LIN {X 0,Y 523.945,Z 504.224,A -85,B 0,C 180,E1 -4885.419,E2 -4885.419} C_VEL
LIN {X 0,Y 523.961,Z 504.216,A -85,B 0,C 180,E1 -4887.999,E2 -4887.999} C_VEL
LIN {X 0,Y 523.943,Z 504.222,A -85,B 0,C 180,E1 -4890.857,E2 -4890.857} C_VEL
LIN {X 0,Y 524,Z 504.295,A -85,B 0,C 180,E1 -4893.743,E2 -4893.743} C_VEL
LIN {X 0,Y 524.381,Z 507.648,A -85,B 0,C 180,E1 -4894.482,E2 -4894.482} C_VEL
LIN {X 0,Y 524.137,Z 518.874,A -85,B 0,C 180,E1 -4896.905,E2 -4896.905} C_VEL
LIN {X 0,Y 525.983,Z 529.654,A -85,B 0,C 180,E1 -4897.12,E2 -4897.12} C_VEL
LIN {X 0,Y 525.614,Z 604.892,A -85,B 0,C 180,E1 -4898.152,E2 -4898.152} C_VEL
LIN {X 0,Y 524.967,Z 610.73,A -85,B 0,C 180,E1 -4898.214,E2 -4898.214} C_VEL
LIN {X 0,Y 519.34,Z 629.652,A -85,B 0,C 180,E1 -4898.382,E2 -4898.382} C_VEL
LIN {X 0,Y 518.506,Z 635.385,A -85,B 0,C 180,E1 -4898.513,E2 -4898.513} C_VEL
LIN {X 0,Y 518.253,Z 648.027,A -85,B 0,C 180,E1 -4898.968,E2 -4898.968} C_VEL
LIN {X 0,Y 517.987,Z 659.606,A -85,B 0,C 180,E1 -4899.537,E2 -4899.537} C_VEL
LIN {X 0,Y 517.725,Z 670.589,A -85,B 0,C 180,E1 -4900.234,E2 -4900.234} C_VEL
LIN {X 0,Y 517.389,Z 681.214,A -85,B 0,C 180,E1 -4901.079,E2 -4901.079} C_VEL
LIN {X 0,Y 517.094,Z 690.566,A -85,B 0,C 180,E1 -4902.002,E2 -4902.002} C_VEL
LIN {X 0,Y 516.862,Z 699.506,A -85,B 0,C 180,E1 -4903.086,E2 -4903.086} C_VEL
LIN {X 0,Y 516.642,Z 706.907,A -85,B 0,C 180,E1 -4904.187,E2 -4904.187} C_VEL
LIN {X 0,Y 516.464,Z 714.132,A -85,B 0,C 180,E1 -4905.541,E2 -4905.541} C_VEL
LIN {X 0,Y 516.394,Z 718.741,A -85,B 0,C 180,E1 -4906.638,E2 -4906.638} C_VEL
LIN {X 0,Y 516.329,Z 722.395,A -85,B 0,C 180,E1 -4907.739,E2 -4907.739} C_VEL
LIN {X 0,Y 516.211,Z 725.817,A -85,B 0,C 180,E1 -4909.195,E2 -4909.195} C_VEL
LIN {X 0,Y 516.162,Z 727.383,A -85,B 0,C 180,E1 -4910.213,E2 -4910.213} C_VEL
LIN {X 0,Y 516.132,Z 728.224,A -85,B 0,C 180,E1 -4911.219,E2 -4911.219} C_VEL
LIN {X 0,Y 516.157,Z 728.432,A -85,B 0,C 180,E1 -4912.215,E2 -4912.215} C_VEL
LIN {X 0,Y 516.162,Z 727.807,A -85,B 0,C 180,E1 -4913.449,E2 -4913.449} C_VEL
LIN {X 0,Y 516.18,Z 726.02,A -85,B 0,C 180,E1 -4914.777,E2 -4914.777} C_VEL
LIN {X 0,Y 516.291,Z 722.961,A -85,B 0,C 180,E1 -4916.135,E2 -4916.135} C_VEL
LIN {X 0,Y 516.389,Z 718.385,A -85,B 0,C 180,E1 -4917.544,E2 -4917.544} C_VEL
LIN {X 0,Y 516.513,Z 712.566,A -85,B 0,C 180,E1 -4918.866,E2 -4918.866} C_VEL
LIN {X 0,Y 516.728,Z 705.121,A -85,B 0,C 180,E1 -4920.183,E2 -4920.183} C_VEL
LIN {X 0,Y 516.932,Z 696.702,A -85,B 0,C 180,E1 -4921.365,E2 -4921.365} C_VEL
LIN {X 0,Y 517.239,Z 686.68,A -85,B 0,C 180,E1 -4922.486,E2 -4922.486} C_VEL
LIN {X 0,Y 517.514,Z 676.852,A -85,B 0,C 180,E1 -4923.376,E2 -4923.376} C_VEL
LIN {X 0,Y 517.839,Z 665.892,A -85,B 0,C 180,E1 -4924.17,E2 -4924.17} C_VEL
LIN {X 0,Y 518.14,Z 653.517,A -85,B 0,C 180,E1 -4924.868,E2 -4924.868} C_VEL
LIN {X 0,Y 518.396,Z 641.103,A -85,B 0,C 180,E1 -4925.39,E2 -4925.39} C_VEL
LIN {X 0,Y 518.587,Z 628.298,A -85,B 0,C 180,E1 -4925.757,E2 -4925.757} C_VEL
LIN {X 0,Y 518.739,Z 608.806,A -85,B 0,C 180,E1 -4926.072,E2 -4926.072} C_VEL
LIN {X 0,Y 519.065,Z 529.137,A -85,B 0,C 180,E1 -4927.182,E2 -4927.182} C_VEL
LIN {X 0,Y 517.13,Z 519.018,A -85,B 0,C 180,E1 -4927.402,E2 -4927.402} C_VEL
LIN {X 0,Y 517.309,Z 507.574,A -85,B 0,C 180,E1 -4929.877,E2 -4929.877} C_VEL
LIN {X 0,Y 516.971,Z 505.092,A -85,B 0,C 180,E1 -4930.442,E2 -4930.442} C_VEL
LIN {X 0,Y 516.911,Z 505.095,A -85,B 0,C 180,E1 -4933.411,E2 -4933.411} C_VEL
LIN {X 0,Y 516.892,Z 505.093,A -85,B 0,C 180,E1 -4935.834,E2 -4935.834} C_VEL
LIN {X 0,Y 516.962,Z 505.086,A -85,B 0,C 180,E1 -4938.234,E2 -4938.234} C_VEL
LIN {X 0,Y 516.966,Z 505.086,A -85,B 0,C 180,E1 -4941.4,E2 -4941.4} C_VEL
LIN {X 0,Y 517,Z 505.08,A -85,B 0,C 180,E1 -4943.757,E2 -4943.757} C_VEL
LIN {X 0,Y 517.012,Z 505.088,A -85,B 0,C 180,E1 -4946.883,E2 -4946.883} C_VEL
LIN {X 0,Y 517.083,Z 505.069,A -85,B 0,C 180,E1 -4950,E2 -4950} C_VEL
LIN {X 0,Y 517.011,Z 505.085,A -85,B 0,C 180,E1 -4953.117,E2 -4953.117} C_VEL
LIN {X 0,Y 517.013,Z 505.079,A -85,B 0,C 180,E1 -4956.243,E2 -4956.243} C_VEL
LIN {X 0,Y 516.952,Z 505.089,A -85,B 0,C 180,E1 -4959.389,E2 -4959.389} C_VEL
LIN {X 0,Y 516.95,Z 505.086,A -85,B 0,C 180,E1 -4961.807,E2 -4961.807} C_VEL
LIN {X 0,Y 516.941,Z 505.094,A -85,B 0,C 180,E1 -4965.146,E2 -4965.146} C_VEL
LIN {X 0,Y 516.923,Z 505.09,A -85,B 0,C 180,E1 -4968.222,E2 -4968.222} C_VEL
LIN {X 0,Y 516.909,Z 505.096,A -85,B 0,C 180,E1 -4970.701,E2 -4970.701} C_VEL
LIN {X 0,Y 516.907,Z 505.091,A -85,B 0,C 180,E1 -4974.072,E2 -4974.072} C_VEL
LIN {X 0,Y 516.922,Z 505.094,A -85,B 0,C 180,E1 -4976.657,E2 -4976.657} C_VEL
LIN {X 0,Y 516.92,Z 505.092,A -85,B 0,C 180,E1 -4979.526,E2 -4979.526} C_VEL
LIN {X 0,Y 516.895,Z 505.095,A -85,B 0,C 180,E1 -4982.544,E2 -4982.544} C_VEL
LIN {X 0,Y 516.877,Z 505.1,A -85,B 0,C 180,E1 -4985.332,E2 -4985.332} C_VEL
LIN {X 0,Y 516.879,Z 505.095,A -85,B 0,C 180,E1 -4987.944,E2 -4987.944} C_VEL
LIN {X 0,Y 516.902,Z 505.097,A -85,B 0,C 180,E1 -4990.739,E2 -4990.739} C_VEL
LIN {X 0,Y 516.876,Z 505.095,A -85,B 0,C 180,E1 -4993.903,E2 -4993.903} C_VEL
LIN {X 0,Y 516.874,Z 505.095,A -85,B 0,C 180,E1 -4996.106,E2 -4996.106} C_VEL
LIN {X 0,Y 516.896,Z 505.099,A -85,B 0,C 180,E1 -4999.26,E2 -4999.26} C_VEL
LIN {X 0,Y 516.877,Z 505.095,A -85,B 0,C 180,E1 -5002.056,E2 -5002.056} C_VEL
LIN {X 0,Y 516.888,Z 505.102,A -85,B 0,C 180,E1 -5005.176,E2 -5005.176} C_VEL
LIN {X 0,Y 516.873,Z 505.096,A -85,B 0,C 180,E1 -5007.976,E2 -5007.976} C_VEL
LIN {X 0,Y 516.926,Z 505.092,A -85,B 0,C 180,E1 -5010.696,E2 -5010.696} C_VEL
LIN {X 0,Y 516.935,Z 505.089,A -85,B 0,C 180,E1 -5013.803,E2 -5013.803} C_VEL
LIN {X 0,Y 516.862,Z 505.101,A -85,B 0,C 180,E1 -5016.777,E2 -5016.777} C_VEL
LIN {X 0,Y 516.929,Z 505.09,A -85,B 0,C 180,E1 -5019.731,E2 -5019.731} C_VEL
LIN {X 0,Y 516.921,Z 505.091,A -85,B 0,C 180,E1 -5022.596,E2 -5022.596} C_VEL
LIN {X 0,Y 516.931,Z 505.096,A -85,B 0,C 180,E1 -5025.03,E2 -5025.03} C_VEL
LIN {X 0,Y 516.994,Z 505.081,A -85,B 0,C 180,E1 -5028.235,E2 -5028.235} C_VEL
LIN {X 0,Y 516.963,Z 505.09,A -85,B 0,C 180,E1 -5031.4,E2 -5031.4} C_VEL
LIN {X 0,Y 517.055,Z 505.074,A -85,B 0,C 180,E1 -5034.541,E2 -5034.541} C_VEL
LIN {X 0,Y 517.075,Z 505.073,A -85,B 0,C 180,E1 -5037.663,E2 -5037.663} C_VEL
LIN {X 0,Y 517.087,Z 505.072,A -85,B 0,C 180,E1 -5040.779,E2 -5040.779} C_VEL
LIN {X 0,Y 517.036,Z 505.083,A -85,B 0,C 180,E1 -5043.117,E2 -5043.117} C_VEL
LIN {X 0,Y 517.007,Z 505.079,A -85,B 0,C 180,E1 -5046.244,E2 -5046.244} C_VEL
LIN {X 0,Y 516.951,Z 505.093,A -85,B 0,C 180,E1 -5049.39,E2 -5049.39} C_VEL
LIN {X 0,Y 516.948,Z 505.088,A -85,B 0,C 180,E1 -5051.811,E2 -5051.811} C_VEL
LIN {X 0,Y 516.935,Z 505.096,A -85,B 0,C 180,E1 -5055.147,E2 -5055.147} C_VEL
LIN {X 0,Y 516.918,Z 505.09,A -85,B 0,C 180,E1 -5058.223,E2 -5058.223} C_VEL
LIN {X 0,Y 516.905,Z 505.093,A -85,B 0,C 180,E1 -5060.702,E2 -5060.702} C_VEL
LIN {X 0,Y 516.904,Z 505.092,A -85,B 0,C 180,E1 -5064.073,E2 -5064.073} C_VEL
LIN {X 0,Y 516.923,Z 505.091,A -85,B 0,C 180,E1 -5066.658,E2 -5066.658} C_VEL
LIN {X 0,Y 516.918,Z 505.096,A -85,B 0,C 180,E1 -5069.527,E2 -5069.527} C_VEL
LIN {X 0,Y 516.895,Z 505.093,A -85,B 0,C 180,E1 -5072.545,E2 -5072.545} C_VEL
LIN {X 0,Y 516.879,Z 505.104,A -85,B 0,C 180,E1 -5075.333,E2 -5075.333} C_VEL
LIN {X 0,Y 516.88,Z 505.096,A -85,B 0,C 180,E1 -5077.945,E2 -5077.945} C_VEL
LIN {X 0,Y 516.882,Z 505.096,A -85,B 0,C 180,E1 -5080.742,E2 -5080.742} C_VEL
LIN {X 0,Y 516.901,Z 505.094,A -85,B 0,C 180,E1 -5082.83,E2 -5082.83} C_VEL
LIN {X 0,Y 516.919,Z 505.094,A -85,B 0,C 180,E1 -5085.011,E2 -5085.011} C_VEL
LIN {X 0,Y 516.921,Z 505.09,A -85,B 0,C 180,E1 -5088.398,E2 -5088.398} C_VEL
LIN {X 0,Y 516.885,Z 505.102,A -85,B 0,C 180,E1 -5091.286,E2 -5091.286} C_VEL
LIN {X 0,Y 516.886,Z 505.094,A -85,B 0,C 180,E1 -5094.222,E2 -5094.222} C_VEL
LIN {X 0,Y 516.897,Z 505.098,A -85,B 0,C 180,E1 -5097.054,E2 -5097.054} C_VEL
LIN {X 0,Y 516.893,Z 505.099,A -85,B 0,C 180,E1 -5099.797,E2 -5099.797} C_VEL
LIN {X 0,Y 516.928,Z 505.092,A -85,B 0,C 180,E1 -5102.468,E2 -5102.468} C_VEL
LIN {X 0,Y 516.976,Z 505.23,A -85,B 0,C 180,E1 -5104.241,E2 -5104.241} C_VEL
LIN {X 0,Y 518.814,Z 514.974,A -85,B 0,C 180,E1 -5105.835,E2 -5105.835} C_VEL
LIN {X 0,Y 518.489,Z 528.641,A -85,B 0,C 180,E1 -5107.905,E2 -5107.905} C_VEL
LIN {X 0,Y 517.995,Z 548.15,A -85,B 0,C 180,E1 -5110.791,E2 -5110.791} C_VEL
LIN {X 0,Y 517.507,Z 568.945,A -85,B 0,C 180,E1 -5113.836,E2 -5113.836} C_VEL
LIN {X 0,Y 517.393,Z 574.378,A -85,B 0,C 180,E1 -5114.63,E2 -5114.63} C_VEL
LIN {X 0,Y 519.12,Z 586.795,A -85,B 0,C 180,E1 -5114.861,E2 -5114.861} C_VEL
LIN {X 0,Y 518.584,Z 682.754,A -85,B 0,C 180,E1 -5116.206,E2 -5116.206} C_VEL
LIN {X 0,Y 518.371,Z 696.184,A -85,B 0,C 180,E1 -5116.55,E2 -5116.55} C_VEL
LIN {X 0,Y 518.095,Z 709.57,A -85,B 0,C 180,E1 -5117.067,E2 -5117.067} C_VEL
LIN {X 0,Y 517.846,Z 721.086,A -85,B 0,C 180,E1 -5117.675,E2 -5117.675} C_VEL
LIN {X 0,Y 517.534,Z 732.47,A -85,B 0,C 180,E1 -5118.446,E2 -5118.446} C_VEL
LIN {X 0,Y 517.2,Z 742.972,A -85,B 0,C 180,E1 -5119.331,E2 -5119.331} C_VEL
LIN {X 0,Y 516.993,Z 751.565,A -85,B 0,C 180,E1 -5120.217,E2 -5120.217} C_VEL
LIN {X 0,Y 516.763,Z 759.494,A -85,B 0,C 180,E1 -5121.199,E2 -5121.199} C_VEL
LIN {X 0,Y 516.563,Z 767.24,A -85,B 0,C 180,E1 -5122.377,E2 -5122.377} C_VEL
LIN {X 0,Y 516.427,Z 774.381,A -85,B 0,C 180,E1 -5123.75,E2 -5123.75} C_VEL
LIN {X 0,Y 516.314,Z 779.131,A -85,B 0,C 180,E1 -5124.924,E2 -5124.924} C_VEL
LIN {X 0,Y 516.355,Z 782.768,A -85,B 0,C 180,E1 -5126.098,E2 -5126.098} C_VEL
LIN {X 0,Y 516.283,Z 784.638,A -85,B 0,C 180,E1 -5126.879,E2 -5126.879} C_VEL
LIN {X 0,Y 516.26,Z 786.042,A -85,B 0,C 180,E1 -5127.659,E2 -5127.659} C_VEL
LIN {X 0,Y 516.16,Z 787.651,A -85,B 0,C 180,E1 -5129.22,E2 -5129.22} C_VEL
LIN {X 0,Y 516.154,Z 787.868,A -85,B 0,C 180,E1 -5130,E2 -5130} C_VEL
LIN {X 0,Y 516.192,Z 787.042,A -85,B 0,C 180,E1 -5131.56,E2 -5131.56} C_VEL
LIN {X 0,Y 516.26,Z 786.043,A -85,B 0,C 180,E1 -5132.341,E2 -5132.341} C_VEL
LIN {X 0,Y 516.283,Z 784.638,A -85,B 0,C 180,E1 -5133.121,E2 -5133.121} C_VEL
LIN {X 0,Y 516.326,Z 781.683,A -85,B 0,C 180,E1 -5134.293,E2 -5134.293} C_VEL
LIN {X 0,Y 516.384,Z 777.682,A -85,B 0,C 180,E1 -5135.467,E2 -5135.467} C_VEL
LIN {X 0,Y 516.444,Z 772.354,A -85,B 0,C 180,E1 -5136.678,E2 -5136.678} C_VEL
LIN {X 0,Y 516.579,Z 766.048,A -85,B 0,C 180,E1 -5137.819,E2 -5137.819} C_VEL
LIN {X 0,Y 516.809,Z 757.966,A -85,B 0,C 180,E1 -5138.997,E2 -5138.997} C_VEL
LIN {X 0,Y 517.021,Z 749.729,A -85,B 0,C 180,E1 -5139.98,E2 -5139.98} C_VEL
LIN {X 0,Y 517.313,Z 739.687,A -85,B 0,C 180,E1 -5140.964,E2 -5140.964} C_VEL
LIN {X 0,Y 517.631,Z 728.435,A -85,B 0,C 180,E1 -5141.844,E2 -5141.844} C_VEL
LIN {X 0,Y 517.942,Z 717.243,A -85,B 0,C 180,E1 -5142.539,E2 -5142.539} C_VEL
LIN {X 0,Y 518.198,Z 704.93,A -85,B 0,C 180,E1 -5143.13,E2 -5143.13} C_VEL
LIN {X 0,Y 518.447,Z 691.96,A -85,B 0,C 180,E1 -5143.573,E2 -5143.573} C_VEL
LIN {X 0,Y 518.654,Z 679.665,A -85,B 0,C 180,E1 -5143.842,E2 -5143.842} C_VEL
LIN {X 0,Y 519.042,Z 585.382,A -85,B 0,C 180,E1 -5145.159,E2 -5145.159} C_VEL
LIN {X 0,Y 517.381,Z 574.125,A -85,B 0,C 180,E1 -5145.38,E2 -5145.38} C_VEL
LIN {X 0,Y 517.857,Z 552.08,A -85,B 0,C 180,E1 -5148.597,E2 -5148.597} C_VEL
LIN {X 0,Y 518.397,Z 531.131,A -85,B 0,C 180,E1 -5151.68,E2 -5151.68} C_VEL
LIN {X 0,Y 518.776,Z 515.802,A -85,B 0,C 180,E1 -5153.979,E2 -5153.979} C_VEL
LIN {X 0,Y 518.207,Z 511.389,A -85,B 0,C 180,E1 -5154.678,E2 -5154.678} C_VEL
LIN {X 0,Y 516.955,Z 505.092,A -85,B 0,C 180,E1 -5155.733,E2 -5155.733} C_VEL
LIN {X 0,Y 516.92,Z 505.098,A -85,B 0,C 180,E1 -5158.414,E2 -5158.414} C_VEL
LIN {X 0,Y 516.891,Z 505.099,A -85,B 0,C 180,E1 -5161.109,E2 -5161.109} C_VEL
LIN {X 0,Y 516.912,Z 505.095,A -85,B 0,C 180,E1 -5163.966,E2 -5163.966} C_VEL
LIN {X 0,Y 516.882,Z 505.104,A -85,B 0,C 180,E1 -5166.745,E2 -5166.745} C_VEL
LIN {X 0,Y 516.901,Z 505.093,A -85,B 0,C 180,E1 -5169.718,E2 -5169.718} C_VEL
LIN {X 0,Y 516.904,Z 505.1,A -85,B 0,C 180,E1 -5172.76,E2 -5172.76} C_VEL
LIN {X 0,Y 516.919,Z 505.095,A -85,B 0,C 180,E1 -5175.009,E2 -5175.009} C_VEL
LIN {X 0,Y 516.913,Z 505.094,A -85,B 0,C 180,E1 -5178.397,E2 -5178.397} C_VEL
LIN {X 0,Y 516.879,Z 505.098,A -85,B 0,C 180,E1 -5181.284,E2 -5181.284} C_VEL
LIN {X 0,Y 516.886,Z 505.096,A -85,B 0,C 180,E1 -5184.22,E2 -5184.22} C_VEL
LIN {X 0,Y 516.893,Z 505.099,A -85,B 0,C 180,E1 -5187.052,E2 -5187.052} C_VEL
LIN {X 0,Y 516.896,Z 505.093,A -85,B 0,C 180,E1 -5189.796,E2 -5189.796} C_VEL
LIN {X 0,Y 516.924,Z 505.093,A -85,B 0,C 180,E1 -5192.467,E2 -5192.467} C_VEL
LIN {X 0,Y 516.905,Z 505.096,A -85,B 0,C 180,E1 -5195.071,E2 -5195.071} C_VEL
LIN {X 0,Y 516.879,Z 505.099,A -85,B 0,C 180,E1 -5198.462,E2 -5198.462} C_VEL
LIN {X 0,Y 516.9,Z 505.101,A -85,B 0,C 180,E1 -5200.954,E2 -5200.954} C_VEL
LIN {X 0,Y 516.909,Z 505.094,A -85,B 0,C 180,E1 -5203.41,E2 -5203.41} C_VEL
LIN {X 0,Y 516.886,Z 505.094,A -85,B 0,C 180,E1 -5205.833,E2 -5205.833} C_VEL
LIN {X 0,Y 516.956,Z 505.087,A -85,B 0,C 180,E1 -5208.233,E2 -5208.233} C_VEL
LIN {X 0,Y 516.964,Z 505.088,A -85,B 0,C 180,E1 -5211.399,E2 -5211.399} C_VEL
LIN {X 0,Y 517.055,Z 505.075,A -85,B 0,C 180,E1 -5214.54,E2 -5214.54} C_VEL
LIN {X 0,Y 517.075,Z 505.072,A -85,B 0,C 180,E1 -5217.663,E2 -5217.663} C_VEL
LIN {X 0,Y 517.087,Z 505.074,A -85,B 0,C 180,E1 -5220.778,E2 -5220.778} C_VEL
LIN {X 0,Y 517.01,Z 505.086,A -85,B 0,C 180,E1 -5223.117,E2 -5223.117} C_VEL
LIN {X 0,Y 517.006,Z 505.079,A -85,B 0,C 180,E1 -5226.243,E2 -5226.243} C_VEL
LIN {X 0,Y 516.949,Z 505.092,A -85,B 0,C 180,E1 -5229.389,E2 -5229.389} C_VEL
LIN {X 0,Y 516.947,Z 505.088,A -85,B 0,C 180,E1 -5231.81,E2 -5231.81} C_VEL
LIN {X 0,Y 516.933,Z 505.097,A -85,B 0,C 180,E1 -5235.146,E2 -5235.146} C_VEL
LIN {X 0,Y 516.917,Z 505.091,A -85,B 0,C 180,E1 -5238.222,E2 -5238.222} C_VEL
LIN {X 0,Y 516.903,Z 505.096,A -85,B 0,C 180,E1 -5240.701,E2 -5240.701} C_VEL
LIN {X 0,Y 516.901,Z 505.095,A -85,B 0,C 180,E1 -5244.072,E2 -5244.072} C_VEL
LIN {X 0,Y 516.92,Z 505.096,A -85,B 0,C 180,E1 -5246.658,E2 -5246.658} C_VEL
LIN {X 0,Y 516.915,Z 505.098,A -85,B 0,C 180,E1 -5249.527,E2 -5249.527} C_VEL
LIN {X 0,Y 516.894,Z 505.099,A -85,B 0,C 180,E1 -5252.545,E2 -5252.545} C_VEL
LIN {X 0,Y 516.929,Z 505.102,A -85,B 0,C 180,E1 -5253.584,E2 -5253.584} C_VEL
LIN {X 0,Y 517.389,Z 509.488,A -85,B 0,C 180,E1 -5254.565,E2 -5254.565} C_VEL
LIN {X 0,Y 517.176,Z 519.353,A -85,B 0,C 180,E1 -5256.703,E2 -5256.703} C_VEL
LIN {X 0,Y 519.152,Z 530.648,A -85,B 0,C 180,E1 -5256.928,E2 -5256.928} C_VEL
LIN {X 0,Y 518.613,Z 625.517,A -85,B 0,C 180,E1 -5258.271,E2 -5258.271} C_VEL
LIN {X 0,Y 518.506,Z 635.385,A -85,B 0,C 180,E1 -5258.513,E2 -5258.513} C_VEL
LIN {X 0,Y 517.638,Z 641.076,A -85,B 0,C 180,E1 -5258.669,E2 -5258.669} C_VEL
LIN {X 0,Y 514.689,Z 650.202,A -85,B 0,C 180,E1 -5258.953,E2 -5258.953} C_VEL
LIN {X 0,Y 511.77,Z 659.029,A -85,B 0,C 180,E1 -5259.327,E2 -5259.327} C_VEL
LIN {X 0,Y 510.95,Z 664.243,A -85,B 0,C 180,E1 -5259.62,E2 -5259.62} C_VEL
LIN {X 0,Y 510.627,Z 675.597,A -85,B 0,C 180,E1 -5260.423,E2 -5260.423} C_VEL
LIN {X 0,Y 510.328,Z 684.665,A -85,B 0,C 180,E1 -5261.216,E2 -5261.216} C_VEL
LIN {X 0,Y 510.034,Z 693.646,A -85,B 0,C 180,E1 -5262.167,E2 -5262.167} C_VEL
LIN {X 0,Y 509.742,Z 702.705,A -85,B 0,C 180,E1 -5263.358,E2 -5263.358} C_VEL
LIN {X 0,Y 509.546,Z 709.578,A -85,B 0,C 180,E1 -5264.475,E2 -5264.475} C_VEL
LIN {X 0,Y 509.393,Z 716.296,A -85,B 0,C 180,E1 -5265.842,E2 -5265.842} C_VEL
LIN {X 0,Y 509.305,Z 720.697,A -85,B 0,C 180,E1 -5267,E2 -5267} C_VEL
LIN {X 0,Y 509.203,Z 724.905,A -85,B 0,C 180,E1 -5268.511,E2 -5268.511} C_VEL
LIN {X 0,Y 509.11,Z 726.92,A -85,B 0,C 180,E1 -5269.549,E2 -5269.549} C_VEL
LIN {X 0,Y 509.071,Z 728.236,A -85,B 0,C 180,E1 -5270.633,E2 -5270.633} C_VEL
LIN {X 0,Y 509.068,Z 728.847,A -85,B 0,C 180,E1 -5271.898,E2 -5271.898} C_VEL
LIN {X 0,Y 509.072,Z 728.435,A -85,B 0,C 180,E1 -5273.198,E2 -5273.198} C_VEL
LIN {X 0,Y 509.086,Z 726.867,A -85,B 0,C 180,E1 -5274.563,E2 -5274.563} C_VEL
LIN {X 0,Y 509.191,Z 724.115,A -85,B 0,C 180,E1 -5275.907,E2 -5275.907} C_VEL
LIN {X 0,Y 509.285,Z 719.822,A -85,B 0,C 180,E1 -5277.328,E2 -5277.328} C_VEL
LIN {X 0,Y 509.465,Z 713.798,A -85,B 0,C 180,E1 -5278.79,E2 -5278.79} C_VEL
LIN {X 0,Y 509.637,Z 707.267,A -85,B 0,C 180,E1 -5280.008,E2 -5280.008} C_VEL
LIN {X 0,Y 509.848,Z 699.633,A -85,B 0,C 180,E1 -5281.155,E2 -5281.155} C_VEL
LIN {X 0,Y 510.148,Z 690.272,A -85,B 0,C 180,E1 -5282.294,E2 -5282.294} C_VEL
LIN {X 0,Y 510.475,Z 680.23,A -85,B 0,C 180,E1 -5283.273,E2 -5283.273} C_VEL
LIN {X 0,Y 510.806,Z 669.716,A -85,B 0,C 180,E1 -5284.098,E2 -5284.098} C_VEL
LIN {X 0,Y 511.11,Z 658.059,A -85,B 0,C 180,E1 -5284.826,E2 -5284.826} C_VEL
LIN {X 0,Y 511.386,Z 646.447,A -85,B 0,C 180,E1 -5285.38,E2 -5285.38} C_VEL
LIN {X 0,Y 511.613,Z 633.316,A -85,B 0,C 180,E1 -5285.825,E2 -5285.825} C_VEL
LIN {X 0,Y 511.807,Z 620.1,A -85,B 0,C 180,E1 -5286.104,E2 -5286.104} C_VEL
LIN {X 0,Y 512.161,Z 529.548,A -85,B 0,C 180,E1 -5287.39,E2 -5287.39} C_VEL
LIN {X 0,Y 510.139,Z 519.449,A -85,B 0,C 180,E1 -5287.609,E2 -5287.609} C_VEL
LIN {X 0,Y 510.336,Z 509.091,A -85,B 0,C 180,E1 -5289.862,E2 -5289.862} C_VEL
LIN {X 0,Y 509.896,Z 505.974,A -85,B 0,C 180,E1 -5290.579,E2 -5290.579} C_VEL
LIN {X 0,Y 509.881,Z 505.973,A -85,B 0,C 180,E1 -5293.175,E2 -5293.175} C_VEL
LIN {X 0,Y 509.861,Z 505.97,A -85,B 0,C 180,E1 -5295.634,E2 -5295.634} C_VEL
LIN {X 0,Y 509.899,Z 505.965,A -85,B 0,C 180,E1 -5298.123,E2 -5298.123} C_VEL
LIN {X 0,Y 509.912,Z 505.966,A -85,B 0,C 180,E1 -5301.28,E2 -5301.28} C_VEL
LIN {X 0,Y 509.951,Z 505.958,A -85,B 0,C 180,E1 -5303.67,E2 -5303.67} C_VEL
LIN {X 0,Y 509.954,Z 505.966,A -85,B 0,C 180,E1 -5306.84,E2 -5306.84} C_VEL
LIN {X 0,Y 510.061,Z 505.949,A -85,B 0,C 180,E1 -5309.211,E2 -5309.211} C_VEL
LIN {X 0,Y 510.054,Z 505.947,A -85,B 0,C 180,E1 -5312.369,E2 -5312.369} C_VEL
LIN {X 0,Y 509.98,Z 505.956,A -85,B 0,C 180,E1 -5316.329,E2 -5316.329} C_VEL
LIN {X 0,Y 509.914,Z 505.968,A -85,B 0,C 180,E1 -5318.72,E2 -5318.72} C_VEL
LIN {X 0,Y 509.901,Z 505.964,A -85,B 0,C 180,E1 -5321.931,E2 -5321.931} C_VEL
LIN {X 0,Y 509.89,Z 505.97,A -85,B 0,C 180,E1 -5325.242,E2 -5325.242} C_VEL
LIN {X 0,Y 509.885,Z 505.966,A -85,B 0,C 180,E1 -5328.001,E2 -5328.001} C_VEL
LIN {X 0,Y 509.846,Z 505.98,A -85,B 0,C 180,E1 -5331.001,E2 -5331.001} C_VEL
LIN {X 0,Y 509.832,Z 505.974,A -85,B 0,C 180,E1 -5333.563,E2 -5333.563} C_VEL
LIN {X 0,Y 509.907,Z 505.965,A -85,B 0,C 180,E1 -5336.378,E2 -5336.378} C_VEL
LIN {X 0,Y 509.881,Z 505.973,A -85,B 0,C 180,E1 -5338.843,E2 -5338.843} C_VEL
LIN {X 0,Y 509.821,Z 505.976,A -85,B 0,C 180,E1 -5341.589,E2 -5341.589} C_VEL
LIN {X 0,Y 509.847,Z 505.972,A -85,B 0,C 180,E1 -5344.413,E2 -5344.413} C_VEL
LIN {X 0,Y 509.816,Z 505.979,A -85,B 0,C 180,E1 -5347.34,E2 -5347.34} C_VEL
LIN {X 0,Y 509.856,Z 505.971,A -85,B 0,C 180,E1 -5350.379,E2 -5350.379} C_VEL
LIN {X 0,Y 509.834,Z 505.982,A -85,B 0,C 180,E1 -5353.064,E2 -5353.064} C_VEL
LIN {X 0,Y 509.822,Z 505.975,A -85,B 0,C 180,E1 -5355.792,E2 -5355.792} C_VEL
LIN {X 0,Y 509.857,Z 505.972,A -85,B 0,C 180,E1 -5358.575,E2 -5358.575} C_VEL
LIN {X 0,Y 509.849,Z 505.971,A -85,B 0,C 180,E1 -5361.785,E2 -5361.785} C_VEL
LIN {X 0,Y 509.838,Z 505.975,A -85,B 0,C 180,E1 -5364.623,E2 -5364.623} C_VEL
LIN {X 0,Y 509.857,Z 505.973,A -85,B 0,C 180,E1 -5367.481,E2 -5367.481} C_VEL
LIN {X 0,Y 509.872,Z 505.968,A -85,B 0,C 180,E1 -5370.269,E2 -5370.269} C_VEL
LIN {X 0,Y 509.878,Z 505.974,A -85,B 0,C 180,E1 -5372.944,E2 -5372.944} C_VEL
LIN {X 0,Y 509.861,Z 505.972,A -85,B 0,C 180,E1 -5375.574,E2 -5375.574} C_VEL
LIN {X 0,Y 509.812,Z 505.975,A -85,B 0,C 180,E1 -5378.149,E2 -5378.149} C_VEL
LIN {X 0,Y 509.855,Z 505.973,A -85,B 0,C 180,E1 -5380.682,E2 -5380.682} C_VEL
LIN {X 0,Y 509.877,Z 505.976,A -85,B 0,C 180,E1 -5383.175,E2 -5383.175} C_VEL
LIN {X 0,Y 509.854,Z 505.973,A -85,B 0,C 180,E1 -5385.634,E2 -5385.634} C_VEL
LIN {X 0,Y 509.919,Z 505.967,A -85,B 0,C 180,E1 -5388.875,E2 -5388.875} C_VEL
LIN {X 0,Y 509.942,Z 505.959,A -85,B 0,C 180,E1 -5392.079,E2 -5392.079} C_VEL
LIN {X 0,Y 510.001,Z 505.952,A -85,B 0,C 180,E1 -5394.465,E2 -5394.465} C_VEL
LIN {X 0,Y 510.046,Z 505.949,A -85,B 0,C 180,E1 -5397.631,E2 -5397.631} C_VEL
LIN {X 0,Y 510.057,Z 505.948,A -85,B 0,C 180,E1 -5400.79,E2 -5400.79} C_VEL
LIN {X 0,Y 509.977,Z 505.963,A -85,B 0,C 180,E1 -5403.16,E2 -5403.16} C_VEL
LIN {X 0,Y 509.974,Z 505.955,A -85,B 0,C 180,E1 -5406.33,E2 -5406.33} C_VEL
LIN {X 0,Y 509.911,Z 505.965,A -85,B 0,C 180,E1 -5408.721,E2 -5408.721} C_VEL
LIN {X 0,Y 509.896,Z 505.966,A -85,B 0,C 180,E1 -5411.932,E2 -5411.932} C_VEL
LIN {X 0,Y 509.885,Z 505.976,A -85,B 0,C 180,E1 -5415.242,E2 -5415.242} C_VEL
LIN {X 0,Y 509.88,Z 505.967,A -85,B 0,C 180,E1 -5418.002,E2 -5418.002} C_VEL
LIN {X 0,Y 509.843,Z 505.976,A -85,B 0,C 180,E1 -5421.002,E2 -5421.002} C_VEL
LIN {X 0,Y 509.829,Z 505.978,A -85,B 0,C 180,E1 -5423.564,E2 -5423.564} C_VEL
LIN {X 0,Y 509.907,Z 505.963,A -85,B 0,C 180,E1 -5426.38,E2 -5426.38} C_VEL
LIN {X 0,Y 509.879,Z 505.97,A -85,B 0,C 180,E1 -5428.844,E2 -5428.844} C_VEL
LIN {X 0,Y 509.821,Z 505.979,A -85,B 0,C 180,E1 -5431.591,E2 -5431.591} C_VEL
LIN {X 0,Y 509.849,Z 505.971,A -85,B 0,C 180,E1 -5434.414,E2 -5434.414} C_VEL
LIN {X 0,Y 509.817,Z 505.984,A -85,B 0,C 180,E1 -5437.341,E2 -5437.341} C_VEL
LIN {X 0,Y 509.834,Z 505.972,A -85,B 0,C 180,E1 -5440.383,E2 -5440.383} C_VEL
LIN {X 0,Y 509.836,Z 505.977,A -85,B 0,C 180,E1 -5443.065,E2 -5443.065} C_VEL
LIN {X 0,Y 509.828,Z 505.976,A -85,B 0,C 180,E1 -5445.793,E2 -5445.793} C_VEL
LIN {X 0,Y 509.863,Z 505.969,A -85,B 0,C 180,E1 -5448.576,E2 -5448.576} C_VEL
LIN {X 0,Y 509.851,Z 505.974,A -85,B 0,C 180,E1 -5451.787,E2 -5451.787} C_VEL
LIN {X 0,Y 509.842,Z 505.972,A -85,B 0,C 180,E1 -5454.624,E2 -5454.624} C_VEL
LIN {X 0,Y 509.866,Z 505.978,A -85,B 0,C 180,E1 -5457.482,E2 -5457.482} C_VEL
LIN {X 0,Y 509.859,Z 505.972,A -85,B 0,C 180,E1 -5460.274,E2 -5460.274} C_VEL
LIN {X 0,Y 509.886,Z 505.973,A -85,B 0,C 180,E1 -5462.945,E2 -5462.945} C_VEL
LIN {X 0,Y 509.937,Z 506.123,A -85,B 0,C 180,E1 -5464.051,E2 -5464.051} C_VEL
LIN {X 0,Y 511.851,Z 515.902,A -85,B 0,C 180,E1 -5465.675,E2 -5465.675} C_VEL
LIN {X 0,Y 511.614,Z 528.317,A -85,B 0,C 180,E1 -5467.593,E2 -5467.593} C_VEL
LIN {X 0,Y 511.018,Z 549.202,A -85,B 0,C 180,E1 -5470.727,E2 -5470.727} C_VEL
LIN {X 0,Y 510.454,Z 569.93,A -85,B 0,C 180,E1 -5473.812,E2 -5473.812} C_VEL
LIN {X 0,Y 510.365,Z 574.163,A -85,B 0,C 180,E1 -5474.419,E2 -5474.419} C_VEL
LIN {X 0,Y 512.249,Z 587.055,A -85,B 0,C 180,E1 -5474.663,E2 -5474.663} C_VEL
LIN {X 0,Y 511.688,Z 682.184,A -85,B 0,C 180,E1 -5476.016,E2 -5476.016} C_VEL
LIN {X 0,Y 511.45,Z 695.682,A -85,B 0,C 180,E1 -5476.365,E2 -5476.365} C_VEL
LIN {X 0,Y 511.164,Z 709.095,A -85,B 0,C 180,E1 -5476.888,E2 -5476.888} C_VEL
LIN {X 0,Y 510.866,Z 720.898,A -85,B 0,C 180,E1 -5477.521,E2 -5477.521} C_VEL
LIN {X 0,Y 510.53,Z 732.026,A -85,B 0,C 180,E1 -5478.285,E2 -5478.285} C_VEL
LIN {X 0,Y 510.217,Z 742.539,A -85,B 0,C 180,E1 -5479.183,E2 -5479.183} C_VEL
LIN {X 0,Y 509.929,Z 751.135,A -85,B 0,C 180,E1 -5480.08,E2 -5480.08} C_VEL
LIN {X 0,Y 509.708,Z 759.071,A -85,B 0,C 180,E1 -5481.077,E2 -5481.077} C_VEL
LIN {X 0,Y 509.486,Z 766.823,A -85,B 0,C 180,E1 -5482.271,E2 -5482.271} C_VEL
LIN {X 0,Y 509.325,Z 773.967,A -85,B 0,C 180,E1 -5483.662,E2 -5483.662} C_VEL
LIN {X 0,Y 509.245,Z 778.723,A -85,B 0,C 180,E1 -5484.853,E2 -5484.853} C_VEL
LIN {X 0,Y 509.266,Z 782.36,A -85,B 0,C 180,E1 -5486.043,E2 -5486.043} C_VEL
LIN {X 0,Y 509.201,Z 784.232,A -85,B 0,C 180,E1 -5486.835,E2 -5486.835} C_VEL
LIN {X 0,Y 509.189,Z 785.637,A -85,B 0,C 180,E1 -5487.627,E2 -5487.627} C_VEL
LIN {X 0,Y 509.073,Z 787.245,A -85,B 0,C 180,E1 -5489.209,E2 -5489.209} C_VEL
LIN {X 0,Y 509.066,Z 787.461,A -85,B 0,C 180,E1 -5490,E2 -5490} C_VEL
LIN {X 0,Y 509.112,Z 786.632,A -85,B 0,C 180,E1 -5491.582,E2 -5491.582} C_VEL
LIN {X 0,Y 509.189,Z 785.632,A -85,B 0,C 180,E1 -5492.373,E2 -5492.373} C_VEL
LIN {X 0,Y 509.201,Z 784.222,A -85,B 0,C 180,E1 -5493.165,E2 -5493.165} C_VEL
LIN {X 0,Y 509.218,Z 781.261,A -85,B 0,C 180,E1 -5494.353,E2 -5494.353} C_VEL
LIN {X 0,Y 509.305,Z 777.256,A -85,B 0,C 180,E1 -5495.543,E2 -5495.543} C_VEL
LIN {X 0,Y 509.396,Z 771.55,A -85,B 0,C 180,E1 -5496.844,E2 -5496.844} C_VEL
LIN {X 0,Y 509.538,Z 764.361,A -85,B 0,C 180,E1 -5498.127,E2 -5498.127} C_VEL
LIN {X 0,Y 509.775,Z 756.01,A -85,B 0,C 180,E1 -5499.322,E2 -5499.322} C_VEL
LIN {X 0,Y 510.018,Z 747.449,A -85,B 0,C 180,E1 -5500.319,E2 -5500.319} C_VEL
LIN {X 0,Y 510.427,Z 736.883,A -85,B 0,C 180,E1 -5501.315,E2 -5501.315} C_VEL
LIN {X 0,Y 510.691,Z 726.091,A -85,B 0,C 180,E1 -5502.137,E2 -5502.137} C_VEL
LIN {X 0,Y 511.015,Z 714.956,A -85,B 0,C 180,E1 -5502.813,E2 -5502.813} C_VEL
LIN {X 0,Y 511.329,Z 703.15,A -85,B 0,C 180,E1 -5503.36,E2 -5503.36} C_VEL
LIN {X 0,Y 511.545,Z 689.542,A -85,B 0,C 180,E1 -5503.81,E2 -5503.81} C_VEL
LIN {X 0,Y 511.78,Z 675.86,A -85,B 0,C 180,E1 -5504.082,E2 -5504.082} C_VEL
LIN {X 0,Y 512.112,Z 585.715,A -85,B 0,C 180,E1 -5505.357,E2 -5505.357} C_VEL
LIN {X 0,Y 510.361,Z 573.691,A -85,B 0,C 180,E1 -5505.594,E2 -5505.594} C_VEL
LIN {X 0,Y 510.888,Z 551.622,A -85,B 0,C 180,E1 -5508.861,E2 -5508.861} C_VEL
LIN {X 0,Y 511.437,Z 532.12,A -85,B 0,C 180,E1 -5511.778,E2 -5511.778} C_VEL
LIN {X 0,Y 511.846,Z 516.823,A -85,B 0,C 180,E1 -5514.109,E2 -5514.109} C_VEL
LIN {X 0,Y 510.396,Z 508.38,A -85,B 0,C 180,E1 -5515.486,E2 -5515.486} C_VEL
LIN {X 0,Y 509.926,Z 505.968,A -85,B 0,C 180,E1 -5515.895,E2 -5515.895} C_VEL
LIN {X 0,Y 509.877,Z 505.974,A -85,B 0,C 180,E1 -5518.843,E2 -5518.843} C_VEL
LIN {X 0,Y 509.825,Z 505.977,A -85,B 0,C 180,E1 -5521.589,E2 -5521.589} C_VEL
LIN {X 0,Y 509.853,Z 505.98,A -85,B 0,C 180,E1 -5524.412,E2 -5524.412} C_VEL
LIN {X 0,Y 509.818,Z 505.977,A -85,B 0,C 180,E1 -5527.34,E2 -5527.34} C_VEL
LIN {X 0,Y 509.859,Z 505.975,A -85,B 0,C 180,E1 -5530.379,E2 -5530.379} C_VEL
LIN {X 0,Y 509.837,Z 505.977,A -85,B 0,C 180,E1 -5533.063,E2 -5533.063} C_VEL
LIN {X 0,Y 509.827,Z 505.974,A -85,B 0,C 180,E1 -5535.791,E2 -5535.791} C_VEL
LIN {X 0,Y 509.855,Z 505.976,A -85,B 0,C 180,E1 -5538.574,E2 -5538.574} C_VEL
LIN {X 0,Y 509.848,Z 505.971,A -85,B 0,C 180,E1 -5541.785,E2 -5541.785} C_VEL
LIN {X 0,Y 509.842,Z 505.978,A -85,B 0,C 180,E1 -5544.622,E2 -5544.622} C_VEL
LIN {X 0,Y 509.86,Z 505.971,A -85,B 0,C 180,E1 -5547.48,E2 -5547.48} C_VEL
LIN {X 0,Y 509.875,Z 505.969,A -85,B 0,C 180,E1 -5550.268,E2 -5550.268} C_VEL
LIN {X 0,Y 509.881,Z 505.975,A -85,B 0,C 180,E1 -5552.944,E2 -5552.944} C_VEL
LIN {X 0,Y 509.863,Z 505.968,A -85,B 0,C 180,E1 -5555.573,E2 -5555.573} C_VEL
LIN {X 0,Y 509.843,Z 505.977,A -85,B 0,C 180,E1 -5558.998,E2 -5558.998} C_VEL
LIN {X 0,Y 509.88,Z 505.967,A -85,B 0,C 180,E1 -5561.998,E2 -5561.998} C_VEL
LIN {X 0,Y 509.901,Z 505.972,A -85,B 0,C 180,E1 -5564.818,E2 -5564.818} C_VEL
LIN {X 0,Y 509.897,Z 505.965,A -85,B 0,C 180,E1 -5568.12,E2 -5568.12} C_VEL
LIN {X 0,Y 509.91,Z 505.968,A -85,B 0,C 180,E1 -5571.279,E2 -5571.279} C_VEL
LIN {X 0,Y 509.973,Z 505.955,A -85,B 0,C 180,E1 -5573.67,E2 -5573.67} C_VEL
LIN {X 0,Y 509.951,Z 505.965,A -85,B 0,C 180,E1 -5576.839,E2 -5576.839} C_VEL
LIN {X 0,Y 510.057,Z 505.95,A -85,B 0,C 180,E1 -5579.21,E2 -5579.21} C_VEL
LIN {X 0,Y 510.046,Z 505.948,A -85,B 0,C 180,E1 -5582.369,E2 -5582.369} C_VEL
LIN {X 0,Y 510.002,Z 505.954,A -85,B 0,C 180,E1 -5585.535,E2 -5585.535} C_VEL
LIN {X 0,Y 509.942,Z 505.96,A -85,B 0,C 180,E1 -5587.921,E2 -5587.921} C_VEL
LIN {X 0,Y 509.908,Z 505.971,A -85,B 0,C 180,E1 -5591.125,E2 -5591.125} C_VEL
LIN {X 0,Y 509.854,Z 505.972,A -85,B 0,C 180,E1 -5594.366,E2 -5594.366} C_VEL
LIN {X 0,Y 509.893,Z 505.969,A -85,B 0,C 180,E1 -5597.651,E2 -5597.651} C_VEL
LIN {X 0,Y 509.876,Z 505.969,A -85,B 0,C 180,E1 -5600.402,E2 -5600.402} C_VEL
LIN {X 0,Y 509.826,Z 505.98,A -85,B 0,C 180,E1 -5603.563,E2 -5603.563} C_VEL
LIN {X 0,Y 509.904,Z 505.969,A -85,B 0,C 180,E1 -5606.379,E2 -5606.379} C_VEL
LIN {X 0,Y 509.876,Z 505.975,A -85,B 0,C 180,E1 -5608.844,E2 -5608.844} C_VEL
LIN {X 0,Y 509.818,Z 505.983,A -85,B 0,C 180,E1 -5611.59,E2 -5611.59} C_VEL
LIN {X 0,Y 509.896,Z 506.076,A -85,B 0,C 180,E1 -5613.458,E2 -5613.458} C_VEL
LIN {X 0,Y 510.416,Z 511.163,A -85,B 0,C 180,E1 -5614.609,E2 -5614.609} C_VEL
LIN {X 0,Y 510.219,Z 519.801,A -85,B 0,C 180,E1 -5616.489,E2 -5616.489} C_VEL
LIN {X 0,Y 512.301,Z 530.6,A -85,B 0,C 180,E1 -5616.716,E2 -5616.716} C_VEL
LIN {X 0,Y 511.74,Z 625.853,A -85,B 0,C 180,E1 -5618.084,E2 -5618.084} C_VEL
LIN {X 0,Y 511.498,Z 639.488,A -85,B 0,C 180,E1 -5618.449,E2 -5618.449} C_VEL
LIN {X 0,Y 511.303,Z 652.192,A -85,B 0,C 180,E1 -5618.96,E2 -5618.96} C_VEL
LIN {X 0,Y 510.95,Z 664.243,A -85,B 0,C 180,E1 -5619.62,E2 -5619.62} C_VEL
LIN {X 0,Y 510.098,Z 669.438,A -85,B 0,C 180,E1 -5619.942,E2 -5619.942} C_VEL
LIN {X 0,Y 507.034,Z 677.595,A -85,B 0,C 180,E1 -5620.486,E2 -5620.486} C_VEL
LIN {X 0,Y 504.004,Z 685.249,A -85,B 0,C 180,E1 -5621.101,E2 -5621.101} C_VEL
LIN {X 0,Y 503.191,Z 689.621,A -85,B 0,C 180,E1 -5621.531,E2 -5621.531} C_VEL
LIN {X 0,Y 502.923,Z 698.265,A -85,B 0,C 180,E1 -5622.557,E2 -5622.557} C_VEL
LIN {X 0,Y 502.635,Z 706.313,A -85,B 0,C 180,E1 -5623.735,E2 -5623.735} C_VEL
LIN {X 0,Y 502.417,Z 713.452,A -85,B 0,C 180,E1 -5625.041,E2 -5625.041} C_VEL
LIN {X 0,Y 502.322,Z 718.354,A -85,B 0,C 180,E1 -5626.169,E2 -5626.169} C_VEL
LIN {X 0,Y 502.219,Z 722.133,A -85,B 0,C 180,E1 -5627.259,E2 -5627.259} C_VEL
LIN {X 0,Y 502.152,Z 725.119,A -85,B 0,C 180,E1 -5628.372,E2 -5628.372} C_VEL
LIN {X 0,Y 502.021,Z 727.88,A -85,B 0,C 180,E1 -5629.913,E2 -5629.913} C_VEL
LIN {X 0,Y 501.982,Z 728.897,A -85,B 0,C 180,E1 -5630.949,E2 -5630.949} C_VEL
LIN {X 0,Y 501.981,Z 729.269,A -85,B 0,C 180,E1 -5631.975,E2 -5631.975} C_VEL
LIN {X 0,Y 501.998,Z 728.977,A -85,B 0,C 180,E1 -5632.988,E2 -5632.988} C_VEL
LIN {X 0,Y 501.991,Z 727.7,A -85,B 0,C 180,E1 -5634.292,E2 -5634.292} C_VEL
LIN {X 0,Y 502.101,Z 725.184,A -85,B 0,C 180,E1 -5635.672,E2 -5635.672} C_VEL
LIN {X 0,Y 502.214,Z 721.257,A -85,B 0,C 180,E1 -5637.101,E2 -5637.101} C_VEL
LIN {X 0,Y 502.372,Z 715.557,A -85,B 0,C 180,E1 -5638.579,E2 -5638.579} C_VEL
LIN {X 0,Y 502.546,Z 709.623,A -85,B 0,C 180,E1 -5639.772,E2 -5639.772} C_VEL
LIN {X 0,Y 502.768,Z 702.442,A -85,B 0,C 180,E1 -5640.939,E2 -5640.939} C_VEL
LIN {X 0,Y 503.061,Z 693.63,A -85,B 0,C 180,E1 -5642.096,E2 -5642.096} C_VEL
LIN {X 0,Y 503.45,Z 683.3,A -85,B 0,C 180,E1 -5643.18,E2 -5643.18} C_VEL
LIN {X 0,Y 503.764,Z 673.134,A -85,B 0,C 180,E1 -5644.043,E2 -5644.043} C_VEL
LIN {X 0,Y 504.12,Z 661.807,A -85,B 0,C 180,E1 -5644.807,E2 -5644.807} C_VEL
LIN {X 0,Y 504.445,Z 649.164,A -85,B 0,C 180,E1 -5645.459,E2 -5645.459} C_VEL
LIN {X 0,Y 504.738,Z 636.293,A -85,B 0,C 180,E1 -5645.939,E2 -5645.939} C_VEL
LIN {X 0,Y 504.901,Z 623.219,A -85,B 0,C 180,E1 -5646.25,E2 -5646.25} C_VEL
LIN {X 0,Y 505.417,Z 531.155,A -85,B 0,C 180,E1 -5647.582,E2 -5647.582} C_VEL
LIN {X 0,Y 503.22,Z 519.746,A -85,B 0,C 180,E1 -5647.847,E2 -5647.847} C_VEL
LIN {X 0,Y 503.32,Z 509.97,A -85,B 0,C 180,E1 -5649.996,E2 -5649.996} C_VEL
LIN {X 0,Y 502.866,Z 506.85,A -85,B 0,C 180,E1 -5650.721,E2 -5650.721} C_VEL
LIN {X 0,Y 502.819,Z 506.848,A -85,B 0,C 180,E1 -5653.767,E2 -5653.767} C_VEL
LIN {X 0,Y 502.832,Z 506.846,A -85,B 0,C 180,E1 -5656.255,E2 -5656.255} C_VEL
LIN {X 0,Y 502.874,Z 506.846,A -85,B 0,C 180,E1 -5658.717,E2 -5658.717} C_VEL
LIN {X 0,Y 502.899,Z 506.836,A -85,B 0,C 180,E1 -5661.967,E2 -5661.967} C_VEL
LIN {X 0,Y 502.931,Z 506.835,A -85,B 0,C 180,E1 -5664.387,E2 -5664.387} C_VEL
LIN {X 0,Y 503.023,Z 506.822,A -85,B 0,C 180,E1 -5667.598,E2 -5667.598} C_VEL
LIN {X 0,Y 503.025,Z 506.821,A -85,B 0,C 180,E1 -5670,E2 -5670} C_VEL
LIN {X 0,Y 503.023,Z 506.823,A -85,B 0,C 180,E1 -5672.402,E2 -5672.402} C_VEL
LIN {X 0,Y 502.939,Z 506.832,A -85,B 0,C 180,E1 -5675.613,E2 -5675.613} C_VEL
LIN {X 0,Y 502.899,Z 506.836,A -85,B 0,C 180,E1 -5678.033,E2 -5678.033} C_VEL
LIN {X 0,Y 502.875,Z 506.844,A -85,B 0,C 180,E1 -5681.283,E2 -5681.283} C_VEL
LIN {X 0,Y 502.842,Z 506.847,A -85,B 0,C 180,E1 -5684.571,E2 -5684.571} C_VEL
LIN {X 0,Y 502.859,Z 506.841,A -85,B 0,C 180,E1 -5687.907,E2 -5687.907} C_VEL
LIN {X 0,Y 502.824,Z 506.849,A -85,B 0,C 180,E1 -5690.536,E2 -5690.536} C_VEL
LIN {X 0,Y 502.793,Z 506.858,A -85,B 0,C 180,E1 -5693.04,E2 -5693.04} C_VEL
LIN {X 0,Y 502.836,Z 506.845,A -85,B 0,C 180,E1 -5695.675,E2 -5695.675} C_VEL
LIN {X 0,Y 502.837,Z 506.845,A -85,B 0,C 180,E1 -5698.372,E2 -5698.372} C_VEL
LIN {X 0,Y 502.792,Z 506.852,A -85,B 0,C 180,E1 -5701.499,E2 -5701.499} C_VEL
LIN {X 0,Y 502.8,Z 506.85,A -85,B 0,C 180,E1 -5704.444,E2 -5704.444} C_VEL
LIN {X 0,Y 502.778,Z 506.858,A -85,B 0,C 180,E1 -5707.178,E2 -5707.178} C_VEL
LIN {X 0,Y 502.82,Z 506.846,A -85,B 0,C 180,E1 -5710.011,E2 -5710.011} C_VEL
LIN {X 0,Y 502.82,Z 506.846,A -85,B 0,C 180,E1 -5712.202,E2 -5712.202} C_VEL
LIN {X 0,Y 502.792,Z 506.853,A -85,B 0,C 180,E1 -5715.468,E2 -5715.468} C_VEL
LIN {X 0,Y 502.821,Z 506.846,A -85,B 0,C 180,E1 -5717.864,E2 -5717.864} C_VEL
LIN {X 0,Y 502.813,Z 506.856,A -85,B 0,C 180,E1 -5721.026,E2 -5721.026} C_VEL
LIN {X 0,Y 502.778,Z 506.851,A -85,B 0,C 180,E1 -5724.167,E2 -5724.167} C_VEL
LIN {X 0,Y 502.824,Z 506.853,A -85,B 0,C 180,E1 -5726.993,E2 -5726.993} C_VEL
LIN {X 0,Y 502.821,Z 506.846,A -85,B 0,C 180,E1 -5730.061,E2 -5730.061} C_VEL
LIN {X 0,Y 502.826,Z 506.847,A -85,B 0,C 180,E1 -5732.533,E2 -5732.533} C_VEL
LIN {X 0,Y 502.819,Z 506.853,A -85,B 0,C 180,E1 -5735.298,E2 -5735.298} C_VEL
LIN {X 0,Y 502.783,Z 506.852,A -85,B 0,C 180,E1 -5737.827,E2 -5737.827} C_VEL
LIN {X 0,Y 502.816,Z 506.847,A -85,B 0,C 180,E1 -5740.4,E2 -5740.4} C_VEL
LIN {X 0,Y 502.826,Z 506.851,A -85,B 0,C 180,E1 -5742.932,E2 -5742.932} C_VEL
LIN {X 0,Y 502.834,Z 506.849,A -85,B 0,C 180,E1 -5745.429,E2 -5745.429} C_VEL
LIN {X 0,Y 502.887,Z 506.841,A -85,B 0,C 180,E1 -5748.717,E2 -5748.717} C_VEL
LIN {X 0,Y 502.892,Z 506.838,A -85,B 0,C 180,E1 -5751.967,E2 -5751.967} C_VEL
LIN {X 0,Y 502.953,Z 506.83,A -85,B 0,C 180,E1 -5754.387,E2 -5754.387} C_VEL
LIN {X 0,Y 503.016,Z 506.825,A -85,B 0,C 180,E1 -5757.598,E2 -5757.598} C_VEL
LIN {X 0,Y 503.017,Z 506.822,A -85,B 0,C 180,E1 -5760,E2 -5760} C_VEL
LIN {X 0,Y 503.019,Z 506.822,A -85,B 0,C 180,E1 -5762.403,E2 -5762.403} C_VEL
LIN {X 0,Y 502.955,Z 506.833,A -85,B 0,C 180,E1 -5765.614,E2 -5765.614} C_VEL
LIN {X 0,Y 502.893,Z 506.837,A -85,B 0,C 180,E1 -5768.034,E2 -5768.034} C_VEL
LIN {X 0,Y 502.873,Z 506.848,A -85,B 0,C 180,E1 -5771.284,E2 -5771.284} C_VEL
LIN {X 0,Y 502.836,Z 506.845,A -85,B 0,C 180,E1 -5774.571,E2 -5774.571} C_VEL
LIN {X 0,Y 502.854,Z 506.843,A -85,B 0,C 180,E1 -5777.908,E2 -5777.908} C_VEL
LIN {X 0,Y 502.82,Z 506.847,A -85,B 0,C 180,E1 -5780.537,E2 -5780.537} C_VEL
LIN {X 0,Y 502.789,Z 506.856,A -85,B 0,C 180,E1 -5783.041,E2 -5783.041} C_VEL
LIN {X 0,Y 502.835,Z 506.848,A -85,B 0,C 180,E1 -5785.676,E2 -5785.676} C_VEL
LIN {X 0,Y 502.836,Z 506.844,A -85,B 0,C 180,E1 -5788.373,E2 -5788.373} C_VEL
LIN {X 0,Y 502.791,Z 506.856,A -85,B 0,C 180,E1 -5791.501,E2 -5791.501} C_VEL
LIN {X 0,Y 502.802,Z 506.849,A -85,B 0,C 180,E1 -5794.446,E2 -5794.446} C_VEL
LIN {X 0,Y 502.778,Z 506.858,A -85,B 0,C 180,E1 -5797.18,E2 -5797.18} C_VEL
LIN {X 0,Y 502.784,Z 506.852,A -85,B 0,C 180,E1 -5800.016,E2 -5800.016} C_VEL
LIN {X 0,Y 502.799,Z 506.849,A -85,B 0,C 180,E1 -5802.2,E2 -5802.2} C_VEL
LIN {X 0,Y 502.798,Z 506.856,A -85,B 0,C 180,E1 -5805.469,E2 -5805.469} C_VEL
LIN {X 0,Y 502.827,Z 506.848,A -85,B 0,C 180,E1 -5807.865,E2 -5807.865} C_VEL
LIN {X 0,Y 502.808,Z 506.852,A -85,B 0,C 180,E1 -5811.026,E2 -5811.026} C_VEL
LIN {X 0,Y 502.781,Z 506.851,A -85,B 0,C 180,E1 -5814.169,E2 -5814.169} C_VEL
LIN {X 0,Y 502.833,Z 506.85,A -85,B 0,C 180,E1 -5816.994,E2 -5816.994} C_VEL
LIN {X 0,Y 502.815,Z 506.851,A -85,B 0,C 180,E1 -5820.066,E2 -5820.066} C_VEL
LIN {X 0,Y 502.834,Z 506.849,A -85,B 0,C 180,E1 -5822.534,E2 -5822.534} C_VEL
LIN {X 0,Y 502.905,Z 507.008,A -85,B 0,C 180,E1 -5823.856,E2 -5823.856} C_VEL
LIN {X 0,Y 505.005,Z 518.371,A -85,B 0,C 180,E1 -5825.762,E2 -5825.762} C_VEL
LIN {X 0,Y 504.413,Z 537.72,A -85,B 0,C 180,E1 -5828.762,E2 -5828.762} C_VEL
LIN {X 0,Y 503.76,Z 557.996,A -85,B 0,C 180,E1 -5831.838,E2 -5831.838} C_VEL
LIN {X 0,Y 503.34,Z 573.596,A -85,B 0,C 180,E1 -5834.19,E2 -5834.19} C_VEL
LIN {X 0,Y 505.369,Z 587.789,A -85,B 0,C 180,E1 -5834.466,E2 -5834.466} C_VEL
LIN {X 0,Y 504.805,Z 681.606,A -85,B 0,C 180,E1 -5835.822,E2 -5835.822} C_VEL
LIN {X 0,Y 504.503,Z 695.177,A -85,B 0,C 180,E1 -5836.173,E2 -5836.173} C_VEL
LIN {X 0,Y 504.249,Z 708.62,A -85,B 0,C 180,E1 -5836.705,E2 -5836.705} C_VEL
LIN {X 0,Y 503.884,Z 720.49,A -85,B 0,C 180,E1 -5837.348,E2 -5837.348} C_VEL
LIN {X 0,Y 503.528,Z 731.582,A -85,B 0,C 180,E1 -5838.12,E2 -5838.12} C_VEL
LIN {X 0,Y 503.152,Z 742.1,A -85,B 0,C 180,E1 -5839.029,E2 -5839.029} C_VEL
LIN {X 0,Y 502.889,Z 750.706,A -85,B 0,C 180,E1 -5839.94,E2 -5839.94} C_VEL
LIN {X 0,Y 502.66,Z 758.649,A -85,B 0,C 180,E1 -5840.95,E2 -5840.95} C_VEL
LIN {X 0,Y 502.406,Z 766.406,A -85,B 0,C 180,E1 -5842.161,E2 -5842.161} C_VEL
LIN {X 0,Y 502.237,Z 773.143,A -85,B 0,C 180,E1 -5843.482,E2 -5843.482} C_VEL
LIN {X 0,Y 502.178,Z 778.314,A -85,B 0,C 180,E1 -5844.781,E2 -5844.781} C_VEL
LIN {X 0,Y 502.16,Z 781.951,A -85,B 0,C 180,E1 -5845.987,E2 -5845.987} C_VEL
LIN {X 0,Y 502.122,Z 783.826,A -85,B 0,C 180,E1 -5846.791,E2 -5846.791} C_VEL
LIN {X 0,Y 502.12,Z 785.232,A -85,B 0,C 180,E1 -5847.594,E2 -5847.594} C_VEL
LIN {X 0,Y 501.99,Z 786.839,A -85,B 0,C 180,E1 -5849.198,E2 -5849.198} C_VEL
LIN {X 0,Y 501.981,Z 787.053,A -85,B 0,C 180,E1 -5850,E2 -5850} C_VEL
LIN {X 0,Y 502.036,Z 786.222,A -85,B 0,C 180,E1 -5851.604,E2 -5851.604} C_VEL
LIN {X 0,Y 502.12,Z 785.22,A -85,B 0,C 180,E1 -5852.406,E2 -5852.406} C_VEL
LIN {X 0,Y 502.122,Z 783.806,A -85,B 0,C 180,E1 -5853.209,E2 -5853.209} C_VEL
LIN {X 0,Y 502.115,Z 780.839,A -85,B 0,C 180,E1 -5854.415,E2 -5854.415} C_VEL
LIN {X 0,Y 502.225,Z 776.829,A -85,B 0,C 180,E1 -5855.621,E2 -5855.621} C_VEL
LIN {X 0,Y 502.331,Z 770.76,A -85,B 0,C 180,E1 -5857.011,E2 -5857.011} C_VEL
LIN {X 0,Y 502.483,Z 763.919,A -85,B 0,C 180,E1 -5858.242,E2 -5858.242} C_VEL
LIN {X 0,Y 502.727,Z 755.557,A -85,B 0,C 180,E1 -5859.454,E2 -5859.454} C_VEL
LIN {X 0,Y 502.993,Z 746.985,A -85,B 0,C 180,E1 -5860.465,E2 -5860.465} C_VEL
LIN {X 0,Y 503.427,Z 736.407,A -85,B 0,C 180,E1 -5861.474,E2 -5861.474} C_VEL
LIN {X 0,Y 503.715,Z 725.601,A -85,B 0,C 180,E1 -5862.308,E2 -5862.308} C_VEL
LIN {X 0,Y 504.065,Z 714.448,A -85,B 0,C 180,E1 -5862.992,E2 -5862.992} C_VEL
LIN {X 0,Y 504.393,Z 702.609,A -85,B 0,C 180,E1 -5863.548,E2 -5863.548} C_VEL
LIN {X 0,Y 504.634,Z 689.877,A -85,B 0,C 180,E1 -5863.977,E2 -5863.977} C_VEL
LIN {X 0,Y 504.881,Z 676.828,A -85,B 0,C 180,E1 -5864.253,E2 -5864.253} C_VEL
LIN {X 0,Y 505.267,Z 586.607,A -85,B 0,C 180,E1 -5865.551,E2 -5865.551} C_VEL
LIN {X 0,Y 503.358,Z 573.16,A -85,B 0,C 180,E1 -5865.829,E2 -5865.829} C_VEL
LIN {X 0,Y 503.924,Z 551.163,A -85,B 0,C 180,E1 -5869.131,E2 -5869.131} C_VEL
LIN {X 0,Y 504.549,Z 530.325,A -85,B 0,C 180,E1 -5872.307,E2 -5872.307} C_VEL
LIN {X 0,Y 504.913,Z 517.843,A -85,B 0,C 180,E1 -5874.243,E2 -5874.243} C_VEL
LIN {X 0,Y 502.863,Z 506.848,A -85,B 0,C 180,E1 -5876.091,E2 -5876.091} C_VEL
LIN {X 0,Y 502.825,Z 506.85,A -85,B 0,C 180,E1 -5879.287,E2 -5879.287} C_VEL
LIN {X 0,Y 502.788,Z 506.856,A -85,B 0,C 180,E1 -5882.083,E2 -5882.083} C_VEL
LIN {X 0,Y 502.809,Z 506.855,A -85,B 0,C 180,E1 -5884.964,E2 -5884.964} C_VEL
LIN {X 0,Y 502.793,Z 506.852,A -85,B 0,C 180,E1 -5887.953,E2 -5887.953} C_VEL
LIN {X 0,Y 502.825,Z 506.851,A -85,B 0,C 180,E1 -5891.064,E2 -5891.064} C_VEL
LIN {X 0,Y 502.779,Z 506.854,A -85,B 0,C 180,E1 -5893.375,E2 -5893.375} C_VEL
LIN {X 0,Y 502.786,Z 506.851,A -85,B 0,C 180,E1 -5895.66,E2 -5895.66} C_VEL
LIN {X 0,Y 502.826,Z 506.845,A -85,B 0,C 180,E1 -5897.863,E2 -5897.863} C_VEL
LIN {X 0,Y 502.798,Z 506.855,A -85,B 0,C 180,E1 -5901.023,E2 -5901.023} C_VEL
LIN {X 0,Y 502.781,Z 506.853,A -85,B 0,C 180,E1 -5904.166,E2 -5904.166} C_VEL
LIN {X 0,Y 502.827,Z 506.852,A -85,B 0,C 180,E1 -5906.992,E2 -5906.992} C_VEL
LIN {X 0,Y 502.824,Z 506.846,A -85,B 0,C 180,E1 -5910.061,E2 -5910.061} C_VEL
LIN {X 0,Y 502.829,Z 506.849,A -85,B 0,C 180,E1 -5912.533,E2 -5912.533} C_VEL
LIN {X 0,Y 502.821,Z 506.847,A -85,B 0,C 180,E1 -5915.298,E2 -5915.298} C_VEL
LIN {X 0,Y 502.773,Z 506.853,A -85,B 0,C 180,E1 -5917.826,E2 -5917.826} C_VEL
LIN {X 0,Y 502.819,Z 506.848,A -85,B 0,C 180,E1 -5920.4,E2 -5920.4} C_VEL
LIN {X 0,Y 502.828,Z 506.851,A -85,B 0,C 180,E1 -5922.931,E2 -5922.931} C_VEL
LIN {X 0,Y 502.836,Z 506.846,A -85,B 0,C 180,E1 -5925.429,E2 -5925.429} C_VEL
LIN {X 0,Y 502.873,Z 506.846,A -85,B 0,C 180,E1 -5928.716,E2 -5928.716} C_VEL
LIN {X 0,Y 502.893,Z 506.838,A -85,B 0,C 180,E1 -5931.966,E2 -5931.966} C_VEL
LIN {X 0,Y 502.954,Z 506.83,A -85,B 0,C 180,E1 -5934.386,E2 -5934.386} C_VEL
LIN {X 0,Y 503.016,Z 506.823,A -85,B 0,C 180,E1 -5937.597,E2 -5937.597} C_VEL
LIN {X 0,Y 503.017,Z 506.821,A -85,B 0,C 180,E1 -5940,E2 -5940} C_VEL
LIN {X 0,Y 503.016,Z 506.824,A -85,B 0,C 180,E1 -5942.402,E2 -5942.402} C_VEL
LIN {X 0,Y 502.954,Z 506.831,A -85,B 0,C 180,E1 -5945.613,E2 -5945.613} C_VEL
LIN {X 0,Y 502.892,Z 506.838,A -85,B 0,C 180,E1 -5948.033,E2 -5948.033} C_VEL
LIN {X 0,Y 502.871,Z 506.847,A -85,B 0,C 180,E1 -5951.283,E2 -5951.283} C_VEL
LIN {X 0,Y 502.835,Z 506.848,A -85,B 0,C 180,E1 -5954.571,E2 -5954.571} C_VEL
LIN {X 0,Y 502.852,Z 506.844,A -85,B 0,C 180,E1 -5957.907,E2 -5957.907} C_VEL
LIN {X 0,Y 502.818,Z 506.849,A -85,B 0,C 180,E1 -5960.536,E2 -5960.536} C_VEL
LIN {X 0,Y 502.786,Z 506.86,A -85,B 0,C 180,E1 -5963.04,E2 -5963.04} C_VEL
LIN {X 0,Y 502.832,Z 506.852,A -85,B 0,C 180,E1 -5965.676,E2 -5965.676} C_VEL
LIN {X 0,Y 502.833,Z 506.849,A -85,B 0,C 180,E1 -5968.373,E2 -5968.373} C_VEL
LIN {X 0,Y 502.788,Z 506.859,A -85,B 0,C 180,E1 -5971.5,E2 -5971.5} C_VEL
LIN {X 0,Y 502.863,Z 506.96,A -85,B 0,C 180,E1 -5973.297,E2 -5973.297} C_VEL
LIN {X 0,Y 503.491,Z 511.045,A -85,B 0,C 180,E1 -5974.245,E2 -5974.245} C_VEL
LIN {X 0,Y 503.312,Z 520.479,A -85,B 0,C 180,E1 -5976.277,E2 -5976.277} C_VEL
LIN {X 0,Y 505.426,Z 531.079,A -85,B 0,C 180,E1 -5976.503,E2 -5976.503} C_VEL
LIN {X 0,Y 504.878,Z 626.304,A -85,B 0,C 180,E1 -5977.895,E2 -5977.895} C_VEL
LIN {X 0,Y 504.625,Z 639.966,A -85,B 0,C 180,E1 -5978.266,E2 -5978.266} C_VEL
LIN {X 0,Y 504.408,Z 652.466,A -85,B 0,C 180,E1 -5978.775,E2 -5978.775} C_VEL
LIN {X 0,Y 504.025,Z 664.925,A -85,B 0,C 180,E1 -5979.468,E2 -5979.468} C_VEL
LIN {X 0,Y 503.667,Z 676.761,A -85,B 0,C 180,E1 -5980.323,E2 -5980.323} C_VEL
LIN {X 0,Y 503.273,Z 687.272,A -85,B 0,C 180,E1 -5981.285,E2 -5981.285} C_VEL
LIN {X 0,Y 503.191,Z 689.621,A -85,B 0,C 180,E1 -5981.531,E2 -5981.531} C_VEL
LIN {X 0,Y 502.381,Z 693.909,A -85,B 0,C 180,E1 -5981.986,E2 -5981.986} C_VEL
LIN {X 0,Y 499.339,Z 700.538,A -85,B 0,C 180,E1 -5982.755,E2 -5982.755} C_VEL
LIN {X 0,Y 496.304,Z 706.532,A -85,B 0,C 180,E1 -5983.595,E2 -5983.595} C_VEL
LIN {X 0,Y 495.513,Z 709.824,A -85,B 0,C 180,E1 -5984.155,E2 -5984.155} C_VEL
LIN {X 0,Y 495.312,Z 716.687,A -85,B 0,C 180,E1 -5985.569,E2 -5985.569} C_VEL
LIN {X 0,Y 495.2,Z 721.023,A -85,B 0,C 180,E1 -5986.714,E2 -5986.714} C_VEL
LIN {X 0,Y 495.088,Z 725.156,A -85,B 0,C 180,E1 -5988.151,E2 -5988.151} C_VEL
LIN {X 0,Y 494.962,Z 727.307,A -85,B 0,C 180,E1 -5989.221,E2 -5989.221} C_VEL
LIN {X 0,Y 494.913,Z 728.756,A -85,B 0,C 180,E1 -5990.282,E2 -5990.282} C_VEL
LIN {X 0,Y 494.917,Z 729.545,A -85,B 0,C 180,E1 -5991.353,E2 -5991.353} C_VEL
LIN {X 0,Y 494.893,Z 729.561,A -85,B 0,C 180,E1 -5992.679,E2 -5992.679} C_VEL
LIN {X 0,Y 494.898,Z 728.488,A -85,B 0,C 180,E1 -5994.041,E2 -5994.041} C_VEL
LIN {X 0,Y 494.997,Z 726.213,A -85,B 0,C 180,E1 -5995.435,E2 -5995.435} C_VEL
LIN {X 0,Y 495.122,Z 722.563,A -85,B 0,C 180,E1 -5996.873,E2 -5996.873} C_VEL
LIN {X 0,Y 495.312,Z 717.304,A -85,B 0,C 180,E1 -5998.357,E2 -5998.357} C_VEL
LIN {X 0,Y 495.477,Z 711.35,A -85,B 0,C 180,E1 -5999.634,E2 -5999.634} C_VEL
LIN {X 0,Y 495.734,Z 703.565,A -85,B 0,C 180,E1 -6000.952,E2 -6000.952} C_VEL
LIN {X 0,Y 496.067,Z 694.921,A -85,B 0,C 180,E1 -6002.127,E2 -6002.127} C_VEL
LIN {X 0,Y 496.44,Z 685.072,A -85,B 0,C 180,E1 -6003.201,E2 -6003.201} C_VEL
LIN {X 0,Y 496.77,Z 674.912,A -85,B 0,C 180,E1 -6004.099,E2 -6004.099} C_VEL
LIN {X 0,Y 497.172,Z 663.441,A -85,B 0,C 180,E1 -6004.908,E2 -6004.908} C_VEL
LIN {X 0,Y 497.493,Z 651.883,A -85,B 0,C 180,E1 -6005.538,E2 -6005.538} C_VEL
LIN {X 0,Y 497.79,Z 638.315,A -85,B 0,C 180,E1 -6006.078,E2 -6006.078} C_VEL
LIN {X 0,Y 498.007,Z 625.705,A -85,B 0,C 180,E1 -6006.409,E2 -6006.409} C_VEL
LIN {X 0,Y 498.602,Z 531.859,A -85,B 0,C 180,E1 -6007.795,E2 -6007.795} C_VEL
LIN {X 0,Y 496.254,Z 520.134,A -85,B 0,C 180,E1 -6008.067,E2 -6008.067} C_VEL
LIN {X 0,Y 496.409,Z 512.728,A -85,B 0,C 180,E1 -6009.705,E2 -6009.705} C_VEL
LIN {X 0,Y 495.798,Z 507.73,A -85,B 0,C 180,E1 -6010.865,E2 -6010.865} C_VEL
LIN {X 0,Y 495.776,Z 507.727,A -85,B 0,C 180,E1 -6013.53,E2 -6013.53} C_VEL
LIN {X 0,Y 495.794,Z 507.722,A -85,B 0,C 180,E1 -6016.056,E2 -6016.056} C_VEL
LIN {X 0,Y 495.849,Z 507.719,A -85,B 0,C 180,E1 -6018.555,E2 -6018.555} C_VEL
LIN {X 0,Y 495.87,Z 507.712,A -85,B 0,C 180,E1 -6021.852,E2 -6021.852} C_VEL
LIN {X 0,Y 495.887,Z 507.711,A -85,B 0,C 180,E1 -6024.307,E2 -6024.307} C_VEL
LIN {X 0,Y 495.992,Z 507.698,A -85,B 0,C 180,E1 -6027.564,E2 -6027.564} C_VEL
LIN {X 0,Y 495.996,Z 507.696,A -85,B 0,C 180,E1 -6030,E2 -6030} C_VEL
LIN {X 0,Y 495.992,Z 507.699,A -85,B 0,C 180,E1 -6032.436,E2 -6032.436} C_VEL
LIN {X 0,Y 495.896,Z 507.709,A -85,B 0,C 180,E1 -6035.693,E2 -6035.693} C_VEL
LIN {X 0,Y 495.871,Z 507.712,A -85,B 0,C 180,E1 -6038.148,E2 -6038.148} C_VEL
LIN {X 0,Y 495.849,Z 507.717,A -85,B 0,C 180,E1 -6041.445,E2 -6041.445} C_VEL
LIN {X 0,Y 495.787,Z 507.729,A -85,B 0,C 180,E1 -6044.783,E2 -6044.783} C_VEL
LIN {X 0,Y 495.783,Z 507.727,A -85,B 0,C 180,E1 -6047.318,E2 -6047.318} C_VEL
LIN {X 0,Y 495.774,Z 507.724,A -85,B 0,C 180,E1 -6049.89,E2 -6049.89} C_VEL
LIN {X 0,Y 495.754,Z 507.734,A -85,B 0,C 180,E1 -6052.86,E2 -6052.86} C_VEL
LIN {X 0,Y 495.786,Z 507.722,A -85,B 0,C 180,E1 -6056.067,E2 -6056.067} C_VEL
LIN {X 0,Y 495.776,Z 507.73,A -85,B 0,C 180,E1 -6058.814,E2 -6058.814} C_VEL
LIN {X 0,Y 495.754,Z 507.727,A -85,B 0,C 180,E1 -6061.726,E2 -6061.726} C_VEL
LIN {X 0,Y 495.77,Z 507.729,A -85,B 0,C 180,E1 -6064.695,E2 -6064.695} C_VEL
LIN {X 0,Y 495.729,Z 507.732,A -85,B 0,C 180,E1 -6067.561,E2 -6067.561} C_VEL
LIN {X 0,Y 495.787,Z 507.722,A -85,B 0,C 180,E1 -6070.052,E2 -6070.052} C_VEL
LIN {X 0,Y 495.757,Z 507.732,A -85,B 0,C 180,E1 -6072.878,E2 -6072.878} C_VEL
LIN {X 0,Y 495.728,Z 507.73,A -85,B 0,C 180,E1 -6075.999,E2 -6075.999} C_VEL
LIN {X 0,Y 495.759,Z 507.729,A -85,B 0,C 180,E1 -6078.705,E2 -6078.705} C_VEL
LIN {X 0,Y 495.756,Z 507.73,A -85,B 0,C 180,E1 -6081.409,E2 -6081.409} C_VEL
LIN {X 0,Y 495.75,Z 507.728,A -85,B 0,C 180,E1 -6084.463,E2 -6084.463} C_VEL
LIN {X 0,Y 495.76,Z 507.73,A -85,B 0,C 180,E1 -6087.406,E2 -6087.406} C_VEL
LIN {X 0,Y 495.772,Z 507.724,A -85,B 0,C 180,E1 -6090.255,E2 -6090.255} C_VEL
LIN {X 0,Y 495.824,Z 507.725,A -85,B 0,C 180,E1 -6093.248,E2 -6093.248} C_VEL
LIN {X 0,Y 495.743,Z 507.729,A -85,B 0,C 180,E1 -6095.725,E2 -6095.725} C_VEL
LIN {X 0,Y 495.737,Z 507.729,A -85,B 0,C 180,E1 -6098.371,E2 -6098.371} C_VEL
LIN {X 0,Y 495.775,Z 507.73,A -85,B 0,C 180,E1 -6100.972,E2 -6100.972} C_VEL
LIN {X 0,Y 495.771,Z 507.728,A -85,B 0,C 180,E1 -6103.53,E2 -6103.53} C_VEL
LIN {X 0,Y 495.784,Z 507.723,A -85,B 0,C 180,E1 -6106.056,E2 -6106.056} C_VEL
LIN {X 0,Y 495.861,Z 507.714,A -85,B 0,C 180,E1 -6108.555,E2 -6108.555} C_VEL
LIN {X 0,Y 495.864,Z 507.714,A -85,B 0,C 180,E1 -6111.852,E2 -6111.852} C_VEL
LIN {X 0,Y 495.907,Z 507.707,A -85,B 0,C 180,E1 -6114.307,E2 -6114.307} C_VEL
LIN {X 0,Y 495.985,Z 507.701,A -85,B 0,C 180,E1 -6117.564,E2 -6117.564} C_VEL
LIN {X 0,Y 495.988,Z 507.698,A -85,B 0,C 180,E1 -6120,E2 -6120} C_VEL
LIN {X 0,Y 495.989,Z 507.698,A -85,B 0,C 180,E1 -6122.437,E2 -6122.437} C_VEL
LIN {X 0,Y 495.909,Z 507.71,A -85,B 0,C 180,E1 -6125.694,E2 -6125.694} C_VEL
LIN {X 0,Y 495.865,Z 507.713,A -85,B 0,C 180,E1 -6128.148,E2 -6128.148} C_VEL
LIN {X 0,Y 495.846,Z 507.721,A -85,B 0,C 180,E1 -6131.446,E2 -6131.446} C_VEL
LIN {X 0,Y 495.781,Z 507.726,A -85,B 0,C 180,E1 -6134.784,E2 -6134.784} C_VEL
LIN {X 0,Y 495.781,Z 507.731,A -85,B 0,C 180,E1 -6137.319,E2 -6137.319} C_VEL
LIN {X 0,Y 495.77,Z 507.726,A -85,B 0,C 180,E1 -6139.891,E2 -6139.891} C_VEL
LIN {X 0,Y 495.758,Z 507.729,A -85,B 0,C 180,E1 -6142.863,E2 -6142.863} C_VEL
LIN {X 0,Y 495.792,Z 507.722,A -85,B 0,C 180,E1 -6146.068,E2 -6146.068} C_VEL
LIN {X 0,Y 495.774,Z 507.726,A -85,B 0,C 180,E1 -6148.815,E2 -6148.815} C_VEL
LIN {X 0,Y 495.753,Z 507.73,A -85,B 0,C 180,E1 -6151.727,E2 -6151.727} C_VEL
LIN {X 0,Y 495.772,Z 507.726,A -85,B 0,C 180,E1 -6154.696,E2 -6154.696} C_VEL
LIN {X 0,Y 495.729,Z 507.735,A -85,B 0,C 180,E1 -6157.562,E2 -6157.562} C_VEL
LIN {X 0,Y 495.763,Z 507.727,A -85,B 0,C 180,E1 -6160.701,E2 -6160.701} C_VEL
LIN {X 0,Y 495.732,Z 507.733,A -85,B 0,C 180,E1 -6163.696,E2 -6163.696} C_VEL
LIN {X 0,Y 495.732,Z 507.729,A -85,B 0,C 180,E1 -6166.306,E2 -6166.306} C_VEL
LIN {X 0,Y 495.778,Z 507.732,A -85,B 0,C 180,E1 -6169.302,E2 -6169.302} C_VEL
LIN {X 0,Y 495.73,Z 507.729,A -85,B 0,C 180,E1 -6172.439,E2 -6172.439} C_VEL
LIN {X 0,Y 495.782,Z 507.731,A -85,B 0,C 180,E1 -6175.458,E2 -6175.458} C_VEL
LIN {X 0,Y 495.759,Z 507.728,A -85,B 0,C 180,E1 -6178.365,E2 -6178.365} C_VEL
LIN {X 0,Y 495.788,Z 507.731,A -85,B 0,C 180,E1 -6181.508,E2 -6181.508} C_VEL
LIN {X 0,Y 495.835,Z 507.75,A -85,B 0,C 180,E1 -6183.629,E2 -6183.629} C_VEL
LIN {X 0,Y 498.057,Z 519.425,A -85,B 0,C 180,E1 -6185.623,E2 -6185.623} C_VEL
LIN {X 0,Y 497.53,Z 536.004,A -85,B 0,C 180,E1 -6188.236,E2 -6188.236} C_VEL
LIN {X 0,Y 496.803,Z 557.329,A -85,B 0,C 180,E1 -6191.532,E2 -6191.532} C_VEL
LIN {X 0,Y 496.316,Z 573.155,A -85,B 0,C 180,E1 -6193.952,E2 -6193.952} C_VEL
LIN {X 0,Y 498.52,Z 589.109,A -85,B 0,C 180,E1 -6194.272,E2 -6194.272} C_VEL
LIN {X 0,Y 497.88,Z 682.261,A -85,B 0,C 180,E1 -6195.647,E2 -6195.647} C_VEL
LIN {X 0,Y 497.584,Z 696.2,A -85,B 0,C 180,E1 -6196.029,E2 -6196.029} C_VEL
LIN {X 0,Y 497.279,Z 709.211,A -85,B 0,C 180,E1 -6196.567,E2 -6196.567} C_VEL
LIN {X 0,Y 496.908,Z 720.476,A -85,B 0,C 180,E1 -6197.197,E2 -6197.197} C_VEL
LIN {X 0,Y 496.486,Z 732.438,A -85,B 0,C 180,E1 -6198.052,E2 -6198.052} C_VEL
LIN {X 0,Y 496.096,Z 742.726,A -85,B 0,C 180,E1 -6198.975,E2 -6198.975} C_VEL
LIN {X 0,Y 495.792,Z 751.978,A -85,B 0,C 180,E1 -6200,E2 -6200} C_VEL
LIN {X 0,Y 495.498,Z 760.987,A -85,B 0,C 180,E1 -6201.23,E2 -6201.23} C_VEL
LIN {X 0,Y 495.286,Z 768.244,A -85,B 0,C 180,E1 -6202.458,E2 -6202.458} C_VEL
LIN {X 0,Y 495.136,Z 774.285,A -85,B 0,C 180,E1 -6203.747,E2 -6203.747} C_VEL
LIN {X 0,Y 495.038,Z 779.227,A -85,B 0,C 180,E1 -6205.114,E2 -6205.114} C_VEL
LIN {X 0,Y 495.056,Z 781.543,A -85,B 0,C 180,E1 -6205.93,E2 -6205.93} C_VEL
LIN {X 0,Y 495.044,Z 783.419,A -85,B 0,C 180,E1 -6206.745,E2 -6206.745} C_VEL
LIN {X 0,Y 495.053,Z 784.828,A -85,B 0,C 180,E1 -6207.559,E2 -6207.559} C_VEL
LIN {X 0,Y 494.911,Z 786.432,A -85,B 0,C 180,E1 -6209.186,E2 -6209.186} C_VEL
LIN {X 0,Y 494.899,Z 786.646,A -85,B 0,C 180,E1 -6210,E2 -6210} C_VEL
LIN {X 0,Y 494.963,Z 785.812,A -85,B 0,C 180,E1 -6211.627,E2 -6211.627} C_VEL
LIN {X 0,Y 495.053,Z 784.807,A -85,B 0,C 180,E1 -6212.441,E2 -6212.441} C_VEL
LIN {X 0,Y 495.044,Z 783.391,A -85,B 0,C 180,E1 -6213.255,E2 -6213.255} C_VEL
LIN {X 0,Y 495.019,Z 780.417,A -85,B 0,C 180,E1 -6214.478,E2 -6214.478} C_VEL
LIN {X 0,Y 495.143,Z 776.402,A -85,B 0,C 180,E1 -6215.702,E2 -6215.702} C_VEL
LIN {X 0,Y 495.257,Z 770.223,A -85,B 0,C 180,E1 -6217.133,E2 -6217.133} C_VEL
LIN {X 0,Y 495.434,Z 763.476,A -85,B 0,C 180,E1 -6218.36,E2 -6218.36} C_VEL
LIN {X 0,Y 495.685,Z 755.105,A -85,B 0,C 180,E1 -6219.59,E2 -6219.59} C_VEL
LIN {X 0,Y 495.981,Z 746.522,A -85,B 0,C 180,E1 -6220.615,E2 -6220.615} C_VEL
LIN {X 0,Y 496.412,Z 735.929,A -85,B 0,C 180,E1 -6221.639,E2 -6221.639} C_VEL
LIN {X 0,Y 496.772,Z 724.414,A -85,B 0,C 180,E1 -6222.533,E2 -6222.533} C_VEL
LIN {X 0,Y 497.132,Z 711.967,A -85,B 0,C 180,E1 -6223.281,E2 -6223.281} C_VEL
LIN {X 0,Y 497.525,Z 699.456,A -85,B 0,C 180,E1 -6223.842,E2 -6223.842} C_VEL
LIN {X 0,Y 497.771,Z 686.479,A -85,B 0,C 180,E1 -6224.252,E2 -6224.252} C_VEL
LIN {X 0,Y 498.042,Z 670.896,A -85,B 0,C 180,E1 -6224.531,E2 -6224.531} C_VEL
LIN {X 0,Y 498.36,Z 586.916,A -85,B 0,C 180,E1 -6225.761,E2 -6225.761} C_VEL
LIN {X 0,Y 496.323,Z 572.711,A -85,B 0,C 180,E1 -6226.058,E2 -6226.058} C_VEL
LIN {X 0,Y 496.921,Z 552.122,A -85,B 0,C 180,E1 -6229.197,E2 -6229.197} C_VEL
LIN {X 0,Y 497.591,Z 531.325,A -85,B 0,C 180,E1 -6232.417,E2 -6232.417} C_VEL
LIN {X 0,Y 497.944,Z 518.835,A -85,B 0,C 180,E1 -6234.382,E2 -6234.382} C_VEL
LIN {X 0,Y 495.818,Z 507.727,A -85,B 0,C 180,E1 -6236.295,E2 -6236.295} C_VEL
LIN {X 0,Y 495.773,Z 507.731,A -85,B 0,C 180,E1 -6238.814,E2 -6238.814} C_VEL
LIN {X 0,Y 495.759,Z 507.73,A -85,B 0,C 180,E1 -6241.725,E2 -6241.725} C_VEL
LIN {X 0,Y 495.776,Z 507.734,A -85,B 0,C 180,E1 -6244.694,E2 -6244.694} C_VEL
LIN {X 0,Y 495.73,Z 507.731,A -85,B 0,C 180,E1 -6247.56,E2 -6247.56} C_VEL
LIN {X 0,Y 495.778,Z 507.731,A -85,B 0,C 180,E1 -6250.698,E2 -6250.698} C_VEL
LIN {X 0,Y 495.732,Z 507.73,A -85,B 0,C 180,E1 -6253.694,E2 -6253.694} C_VEL
LIN {X 0,Y 495.731,Z 507.733,A -85,B 0,C 180,E1 -6256.304,E2 -6256.304} C_VEL
LIN {X 0,Y 495.763,Z 507.728,A -85,B 0,C 180,E1 -6259.299,E2 -6259.299} C_VEL
LIN {X 0,Y 495.729,Z 507.735,A -85,B 0,C 180,E1 -6262.438,E2 -6262.438} C_VEL
LIN {X 0,Y 495.781,Z 507.723,A -85,B 0,C 180,E1 -6265.457,E2 -6265.457} C_VEL
LIN {X 0,Y 495.754,Z 507.73,A -85,B 0,C 180,E1 -6268.363,E2 -6268.363} C_VEL
LIN {X 0,Y 495.784,Z 507.723,A -85,B 0,C 180,E1 -6271.505,E2 -6271.505} C_VEL
LIN {X 0,Y 495.792,Z 507.723,A -85,B 0,C 180,E1 -6273.932,E2 -6273.932} C_VEL
LIN {X 0,Y 495.753,Z 507.732,A -85,B 0,C 180,E1 -6277.138,E2 -6277.138} C_VEL
LIN {X 0,Y 495.771,Z 507.724,A -85,B 0,C 180,E1 -6280.109,E2 -6280.109} C_VEL
LIN {X 0,Y 495.78,Z 507.729,A -85,B 0,C 180,E1 -6282.681,E2 -6282.681} C_VEL
LIN {X 0,Y 495.781,Z 507.727,A -85,B 0,C 180,E1 -6285.216,E2 -6285.216} C_VEL
LIN {X 0,Y 495.846,Z 507.719,A -85,B 0,C 180,E1 -6288.554,E2 -6288.554} C_VEL
LIN {X 0,Y 495.865,Z 507.714,A -85,B 0,C 180,E1 -6291.852,E2 -6291.852} C_VEL
LIN {X 0,Y 495.908,Z 507.707,A -85,B 0,C 180,E1 -6294.306,E2 -6294.306} C_VEL
LIN {X 0,Y 495.985,Z 507.7,A -85,B 0,C 180,E1 -6297.563,E2 -6297.563} C_VEL
LIN {X 0,Y 495.988,Z 507.697,A -85,B 0,C 180,E1 -6300,E2 -6300} C_VEL
LIN {X 0,Y 495.985,Z 507.7,A -85,B 0,C 180,E1 -6302.436,E2 -6302.436} C_VEL
LIN {X 0,Y 495.908,Z 507.708,A -85,B 0,C 180,E1 -6305.693,E2 -6305.693} C_VEL
LIN {X 0,Y 495.864,Z 507.714,A -85,B 0,C 180,E1 -6308.148,E2 -6308.148} C_VEL
LIN {X 0,Y 495.845,Z 507.72,A -85,B 0,C 180,E1 -6311.445,E2 -6311.445} C_VEL
LIN {X 0,Y 495.78,Z 507.729,A -85,B 0,C 180,E1 -6314.783,E2 -6314.783} C_VEL
LIN {X 0,Y 495.778,Z 507.731,A -85,B 0,C 180,E1 -6317.318,E2 -6317.318} C_VEL
LIN {X 0,Y 495.769,Z 507.727,A -85,B 0,C 180,E1 -6319.89,E2 -6319.89} C_VEL
LIN {X 0,Y 495.755,Z 507.733,A -85,B 0,C 180,E1 -6322.862,E2 -6322.862} C_VEL
LIN {X 0,Y 495.789,Z 507.727,A -85,B 0,C 180,E1 -6326.067,E2 -6326.067} C_VEL
LIN {X 0,Y 495.771,Z 507.732,A -85,B 0,C 180,E1 -6328.814,E2 -6328.814} C_VEL
LIN {X 0,Y 495.75,Z 507.735,A -85,B 0,C 180,E1 -6331.726,E2 -6331.726} C_VEL
LIN {X 0,Y 495.812,Z 507.746,A -85,B 0,C 180,E1 -6333.113,E2 -6333.113} C_VEL
LIN {X 0,Y 496.517,Z 512.575,A -85,B 0,C 180,E1 -6334.238,E2 -6334.238} C_VEL
LIN {X 0,Y 496.328,Z 520.655,A -85,B 0,C 180,E1 -6336.045,E2 -6336.045} C_VEL
LIN {X 0,Y 498.635,Z 532.19,A -85,B 0,C 180,E1 -6336.296,E2 -6336.296} C_VEL
LIN {X 0,Y 497.979,Z 627.35,A -85,B 0,C 180,E1 -6337.713,E2 -6337.713} C_VEL
LIN {X 0,Y 497.731,Z 641.206,A -85,B 0,C 180,E1 -6338.104,E2 -6338.104} C_VEL
LIN {X 0,Y 497.494,Z 653.909,A -85,B 0,C 180,E1 -6338.643,E2 -6338.643} C_VEL
LIN {X 0,Y 497.076,Z 666.464,A -85,B 0,C 180,E1 -6339.367,E2 -6339.367} C_VEL
LIN {X 0,Y 496.727,Z 677.436,A -85,B 0,C 180,E1 -6340.181,E2 -6340.181} C_VEL
LIN {X 0,Y 496.298,Z 688.076,A -85,B 0,C 180,E1 -6341.177,E2 -6341.177} C_VEL
LIN {X 0,Y 495.939,Z 697.959,A -85,B 0,C 180,E1 -6342.331,E2 -6342.331} C_VEL
LIN {X 0,Y 495.642,Z 705.888,A -85,B 0,C 180,E1 -6343.478,E2 -6343.478} C_VEL
LIN {X 0,Y 495.513,Z 709.824,A -85,B 0,C 180,E1 -6344.155,E2 -6344.155} C_VEL
LIN {X 0,Y 494.718,Z 712.949,A -85,B 0,C 180,E1 -6344.734,E2 -6344.734} C_VEL
LIN {X 0,Y 491.68,Z 717.614,A -85,B 0,C 180,E1 -6345.691,E2 -6345.691} C_VEL
LIN {X 0,Y 488.736,Z 721.577,A -85,B 0,C 180,E1 -6346.696,E2 -6346.696} C_VEL
LIN {X 0,Y 488.091,Z 723.601,A -85,B 0,C 180,E1 -6347.34,E2 -6347.34} C_VEL
LIN {X 0,Y 487.952,Z 726.456,A -85,B 0,C 180,E1 -6348.507,E2 -6348.507} C_VEL
LIN {X 0,Y 487.853,Z 728.598,A -85,B 0,C 180,E1 -6349.774,E2 -6349.774} C_VEL
LIN {X 0,Y 487.816,Z 729.805,A -85,B 0,C 180,E1 -6351.075,E2 -6351.075} C_VEL
LIN {X 0,Y 487.81,Z 729.935,A -85,B 0,C 180,E1 -6352.765,E2 -6352.765} C_VEL
LIN {X 0,Y 487.803,Z 729.175,A -85,B 0,C 180,E1 -6353.794,E2 -6353.794} C_VEL
LIN {X 0,Y 487.905,Z 727.181,A -85,B 0,C 180,E1 -6355.189,E2 -6355.189} C_VEL
LIN {X 0,Y 488.032,Z 723.855,A -85,B 0,C 180,E1 -6356.64,E2 -6356.64} C_VEL
LIN {X 0,Y 488.187,Z 718.883,A -85,B 0,C 180,E1 -6358.142,E2 -6358.142} C_VEL
LIN {X 0,Y 488.42,Z 712.839,A -85,B 0,C 180,E1 -6359.522,E2 -6359.522} C_VEL
LIN {X 0,Y 488.672,Z 706.194,A -85,B 0,C 180,E1 -6360.727,E2 -6360.727} C_VEL
LIN {X 0,Y 488.973,Z 698.035,A -85,B 0,C 180,E1 -6361.92,E2 -6361.92} C_VEL
LIN {X 0,Y 489.362,Z 688.813,A -85,B 0,C 180,E1 -6363.012,E2 -6363.012} C_VEL
LIN {X 0,Y 489.742,Z 678.046,A -85,B 0,C 180,E1 -6364.044,E2 -6364.044} C_VEL
LIN {X 0,Y 490.171,Z 667.21,A -85,B 0,C 180,E1 -6364.865,E2 -6364.865} C_VEL
LIN {X 0,Y 490.517,Z 655.53,A -85,B 0,C 180,E1 -6365.562,E2 -6365.562} C_VEL
LIN {X 0,Y 490.824,Z 643.591,A -85,B 0,C 180,E1 -6366.101,E2 -6366.101} C_VEL
LIN {X 0,Y 491.057,Z 630.884,A -85,B 0,C 180,E1 -6366.502,E2 -6366.502} C_VEL
LIN {X 0,Y 491.222,Z 614.105,A -85,B 0,C 180,E1 -6366.804,E2 -6366.804} C_VEL
LIN {X 0,Y 491.712,Z 532.339,A -85,B 0,C 180,E1 -6368.02,E2 -6368.02} C_VEL
LIN {X 0,Y 489.306,Z 520.504,A -85,B 0,C 180,E1 -6368.294,E2 -6368.294} C_VEL
LIN {X 0,Y 489.412,Z 513.57,A -85,B 0,C 180,E1 -6369.841,E2 -6369.841} C_VEL
LIN {X 0,Y 488.757,Z 508.607,A -85,B 0,C 180,E1 -6371.015,E2 -6371.015} C_VEL
LIN {X 0,Y 488.773,Z 508.601,A -85,B 0,C 180,E1 -6374.445,E2 -6374.445} C_VEL
LIN {X 0,Y 488.786,Z 508.594,A -85,B 0,C 180,E1 -6377.885,E2 -6377.885} C_VEL
LIN {X 0,Y 488.781,Z 508.604,A -85,B 0,C 180,E1 -6380.9,E2 -6380.9} C_VEL
LIN {X 0,Y 488.815,Z 508.593,A -85,B 0,C 180,E1 -6383.395,E2 -6383.395} C_VEL
LIN {X 0,Y 488.699,Z 508.605,A -85,B 0,C 180,E1 -6385.877,E2 -6385.877} C_VEL
LIN {X 0,Y 488.96,Z 508.574,A -85,B 0,C 180,E1 -6387.529,E2 -6387.529} C_VEL
LIN {X 0,Y 488.952,Z 508.581,A -85,B 0,C 180,E1 -6390.824,E2 -6390.824} C_VEL
LIN {X 0,Y 488.959,Z 508.576,A -85,B 0,C 180,E1 -6392.471,E2 -6392.471} C_VEL
LIN {X 0,Y 488.855,Z 508.586,A -85,B 0,C 180,E1 -6395.776,E2 -6395.776} C_VEL
LIN {X 0,Y 488.815,Z 508.592,A -85,B 0,C 180,E1 -6398.266,E2 -6398.266} C_VEL
LIN {X 0,Y 488.803,Z 508.593,A -85,B 0,C 180,E1 -6401.612,E2 -6401.612} C_VEL
LIN {X 0,Y 488.759,Z 508.607,A -85,B 0,C 180,E1 -6405,E2 -6405} C_VEL
LIN {X 0,Y 488.751,Z 508.601,A -85,B 0,C 180,E1 -6408.442,E2 -6408.442} C_VEL
LIN {X 0,Y 488.704,Z 508.612,A -85,B 0,C 180,E1 -6411.07,E2 -6411.07} C_VEL
LIN {X 0,Y 488.689,Z 508.607,A -85,B 0,C 180,E1 -6413.745,E2 -6413.745} C_VEL
LIN {X 0,Y 488.787,Z 508.603,A -85,B 0,C 180,E1 -6416.943,E2 -6416.943} C_VEL
LIN {X 0,Y 488.729,Z 508.602,A -85,B 0,C 180,E1 -6420.218,E2 -6420.218} C_VEL
LIN {X 0,Y 488.73,Z 508.604,A -85,B 0,C 180,E1 -6423.484,E2 -6423.484} C_VEL
LIN {X 0,Y 488.684,Z 508.608,A -85,B 0,C 180,E1 -6426.356,E2 -6426.356} C_VEL
LIN {X 0,Y 488.742,Z 508.606,A -85,B 0,C 180,E1 -6429.249,E2 -6429.249} C_VEL
LIN {X 0,Y 488.727,Z 508.604,A -85,B 0,C 180,E1 -6432.52,E2 -6432.52} C_VEL
LIN {X 0,Y 488.704,Z 508.612,A -85,B 0,C 180,E1 -6435.198,E2 -6435.198} C_VEL
LIN {X 0,Y 488.727,Z 508.605,A -85,B 0,C 180,E1 -6437.479,E2 -6437.479} C_VEL
LIN {X 0,Y 488.74,Z 508.604,A -85,B 0,C 180,E1 -6440.75,E2 -6440.75} C_VEL
LIN {X 0,Y 488.678,Z 508.608,A -85,B 0,C 180,E1 -6443.869,E2 -6443.869} C_VEL
LIN {X 0,Y 488.73,Z 508.607,A -85,B 0,C 180,E1 -6446.877,E2 -6446.877} C_VEL
LIN {X 0,Y 488.724,Z 508.603,A -85,B 0,C 180,E1 -6449.781,E2 -6449.781} C_VEL
LIN {X 0,Y 488.789,Z 508.602,A -85,B 0,C 180,E1 -6453.055,E2 -6453.055} C_VEL
LIN {X 0,Y 488.684,Z 508.607,A -85,B 0,C 180,E1 -6456.255,E2 -6456.255} C_VEL
LIN {X 0,Y 488.736,Z 508.609,A -85,B 0,C 180,E1 -6459.176,E2 -6459.176} C_VEL
LIN {X 0,Y 488.749,Z 508.602,A -85,B 0,C 180,E1 -6461.628,E2 -6461.628} C_VEL
LIN {X 0,Y 488.751,Z 508.605,A -85,B 0,C 180,E1 -6465,E2 -6465} C_VEL
LIN {X 0,Y 488.822,Z 508.59,A -85,B 0,C 180,E1 -6468.388,E2 -6468.388} C_VEL
LIN {X 0,Y 488.809,Z 508.593,A -85,B 0,C 180,E1 -6471.734,E2 -6471.734} C_VEL
LIN {X 0,Y 488.864,Z 508.585,A -85,B 0,C 180,E1 -6474.225,E2 -6474.225} C_VEL
LIN {X 0,Y 488.953,Z 508.578,A -85,B 0,C 180,E1 -6477.529,E2 -6477.529} C_VEL
LIN {X 0,Y 488.959,Z 508.573,A -85,B 0,C 180,E1 -6480,E2 -6480} C_VEL
LIN {X 0,Y 488.958,Z 508.574,A -85,B 0,C 180,E1 -6482.472,E2 -6482.472} C_VEL
LIN {X 0,Y 488.865,Z 508.586,A -85,B 0,C 180,E1 -6485.776,E2 -6485.776} C_VEL
LIN {X 0,Y 488.81,Z 508.591,A -85,B 0,C 180,E1 -6488.267,E2 -6488.267} C_VEL
LIN {X 0,Y 488.799,Z 508.596,A -85,B 0,C 180,E1 -6491.613,E2 -6491.613} C_VEL
LIN {X 0,Y 488.753,Z 508.604,A -85,B 0,C 180,E1 -6495.001,E2 -6495.001} C_VEL
LIN {X 0,Y 488.747,Z 508.6,A -85,B 0,C 180,E1 -6498.443,E2 -6498.443} C_VEL
LIN {X 0,Y 488.699,Z 508.611,A -85,B 0,C 180,E1 -6501.071,E2 -6501.071} C_VEL
LIN {X 0,Y 488.686,Z 508.61,A -85,B 0,C 180,E1 -6503.746,E2 -6503.746} C_VEL
LIN {X 0,Y 488.792,Z 508.598,A -85,B 0,C 180,E1 -6506.946,E2 -6506.946} C_VEL
LIN {X 0,Y 488.713,Z 508.604,A -85,B 0,C 180,E1 -6510.366,E2 -6510.366} C_VEL
LIN {X 0,Y 488.731,Z 508.608,A -85,B 0,C 180,E1 -6513.485,E2 -6513.485} C_VEL
LIN {X 0,Y 488.685,Z 508.607,A -85,B 0,C 180,E1 -6516.357,E2 -6516.357} C_VEL
LIN {X 0,Y 488.697,Z 508.613,A -85,B 0,C 180,E1 -6519.255,E2 -6519.255} C_VEL
LIN {X 0,Y 488.72,Z 508.608,A -85,B 0,C 180,E1 -6521.603,E2 -6521.603} C_VEL
LIN {X 0,Y 488.709,Z 508.606,A -85,B 0,C 180,E1 -6524.802,E2 -6524.802} C_VEL
LIN {X 0,Y 488.733,Z 508.608,A -85,B 0,C 180,E1 -6527.48,E2 -6527.48} C_VEL
LIN {X 0,Y 488.741,Z 508.601,A -85,B 0,C 180,E1 -6530.751,E2 -6530.751} C_VEL
LIN {X 0,Y 488.682,Z 508.61,A -85,B 0,C 180,E1 -6533.869,E2 -6533.869} C_VEL
LIN {X 0,Y 488.739,Z 508.605,A -85,B 0,C 180,E1 -6536.878,E2 -6536.878} C_VEL
LIN {X 0,Y 488.724,Z 508.608,A -85,B 0,C 180,E1 -6539.782,E2 -6539.782} C_VEL
LIN {X 0,Y 488.793,Z 508.602,A -85,B 0,C 180,E1 -6543.057,E2 -6543.057} C_VEL
LIN {X 0,Y 488.807,Z 508.716,A -85,B 0,C 180,E1 -6543.437,E2 -6543.437} C_VEL
LIN {X 0,Y 491.105,Z 520.469,A -85,B 0,C 180,E1 -6545.481,E2 -6545.481} C_VEL
LIN {X 0,Y 490.807,Z 531.517,A -85,B 0,C 180,E1 -6547.256,E2 -6547.256} C_VEL
LIN {X 0,Y 489.997,Z 553.591,A -85,B 0,C 180,E1 -6550.739,E2 -6550.739} C_VEL
LIN {X 0,Y 489.346,Z 572.819,A -85,B 0,C 180,E1 -6553.726,E2 -6553.726} C_VEL
LIN {X 0,Y 491.669,Z 589.96,A -85,B 0,C 180,E1 -6554.066,E2 -6554.066} C_VEL
LIN {X 0,Y 491.004,Z 681.71,A -85,B 0,C 180,E1 -6555.441,E2 -6555.441} C_VEL
LIN {X 0,Y 490.7,Z 694.934,A -85,B 0,C 180,E1 -6555.803,E2 -6555.803} C_VEL
LIN {X 0,Y 490.395,Z 707.665,A -85,B 0,C 180,E1 -6556.322,E2 -6556.322} C_VEL
LIN {X 0,Y 489.998,Z 718.928,A -85,B 0,C 180,E1 -6556.94,E2 -6556.94} C_VEL
LIN {X 0,Y 489.582,Z 730.696,A -85,B 0,C 180,E1 -6557.776,E2 -6557.776} C_VEL
LIN {X 0,Y 489.193,Z 741.233,A -85,B 0,C 180,E1 -6558.712,E2 -6558.712} C_VEL
LIN {X 0,Y 488.825,Z 749.849,A -85,B 0,C 180,E1 -6559.647,E2 -6559.647} C_VEL
LIN {X 0,Y 488.519,Z 757.8,A -85,B 0,C 180,E1 -6560.686,E2 -6560.686} C_VEL
LIN {X 0,Y 488.275,Z 765.573,A -85,B 0,C 180,E1 -6561.933,E2 -6561.933} C_VEL
LIN {X 0,Y 488.101,Z 772.73,A -85,B 0,C 180,E1 -6563.386,E2 -6563.386} C_VEL
LIN {X 0,Y 488.045,Z 777.496,A -85,B 0,C 180,E1 -6564.629,E2 -6564.629} C_VEL
LIN {X 0,Y 487.952,Z 781.134,A -85,B 0,C 180,E1 -6565.87,E2 -6565.87} C_VEL
LIN {X 0,Y 487.968,Z 783.014,A -85,B 0,C 180,E1 -6566.697,E2 -6566.697} C_VEL
LIN {X 0,Y 487.959,Z 784.421,A -85,B 0,C 180,E1 -6567.524,E2 -6567.524} C_VEL
LIN {X 0,Y 487.893,Z 785.42,A -85,B 0,C 180,E1 -6568.349,E2 -6568.349} C_VEL
LIN {X 0,Y 487.82,Z 786.239,A -85,B 0,C 180,E1 -6570,E2 -6570} C_VEL
LIN {X 0,Y 487.893,Z 785.402,A -85,B 0,C 180,E1 -6571.651,E2 -6571.651} C_VEL
LIN {X 0,Y 487.959,Z 784.393,A -85,B 0,C 180,E1 -6572.476,E2 -6572.476} C_VEL
LIN {X 0,Y 487.968,Z 782.975,A -85,B 0,C 180,E1 -6573.303,E2 -6573.303} C_VEL
LIN {X 0,Y 487.929,Z 779.996,A -85,B 0,C 180,E1 -6574.544,E2 -6574.544} C_VEL
LIN {X 0,Y 488.042,Z 775.974,A -85,B 0,C 180,E1 -6575.785,E2 -6575.785} C_VEL
LIN {X 0,Y 488.183,Z 769.788,A -85,B 0,C 180,E1 -6577.236,E2 -6577.236} C_VEL
LIN {X 0,Y 488.364,Z 763.03,A -85,B 0,C 180,E1 -6578.482,E2 -6578.482} C_VEL
LIN {X 0,Y 488.616,Z 754.65,A -85,B 0,C 180,E1 -6579.73,E2 -6579.73} C_VEL
LIN {X 0,Y 488.971,Z 746.058,A -85,B 0,C 180,E1 -6580.769,E2 -6580.769} C_VEL
LIN {X 0,Y 489.412,Z 735.451,A -85,B 0,C 180,E1 -6581.808,E2 -6581.808} C_VEL
LIN {X 0,Y 489.833,Z 723.662,A -85,B 0,C 180,E1 -6582.733,E2 -6582.733} C_VEL
LIN {X 0,Y 490.178,Z 711.45,A -85,B 0,C 180,E1 -6583.473,E2 -6583.473} C_VEL
LIN {X 0,Y 490.59,Z 698.914,A -85,B 0,C 180,E1 -6584.042,E2 -6584.042} C_VEL
LIN {X 0,Y 490.882,Z 685.867,A -85,B 0,C 180,E1 -6584.457,E2 -6584.457} C_VEL
LIN {X 0,Y 491.168,Z 670.186,A -85,B 0,C 180,E1 -6584.739,E2 -6584.739} C_VEL
LIN {X 0,Y 491.578,Z 588.231,A -85,B 0,C 180,E1 -6585.957,E2 -6585.957} C_VEL
LIN {X 0,Y 489.313,Z 572.309,A -85,B 0,C 180,E1 -6586.287,E2 -6586.287} C_VEL
LIN {X 0,Y 489.966,Z 551.706,A -85,B 0,C 180,E1 -6589.481,E2 -6589.481} C_VEL
LIN {X 0,Y 490.629,Z 532.318,A -85,B 0,C 180,E1 -6592.53,E2 -6592.53} C_VEL
LIN {X 0,Y 491.055,Z 521.243,A -85,B 0,C 180,E1 -6594.297,E2 -6594.297} C_VEL
LIN {X 0,Y 489.944,Z 514.264,A -85,B 0,C 180,E1 -6595.488,E2 -6595.488} C_VEL
LIN {X 0,Y 488.807,Z 508.6,A -85,B 0,C 180,E1 -6596.506,E2 -6596.506} C_VEL
LIN {X 0,Y 488.724,Z 508.607,A -85,B 0,C 180,E1 -6599.27,E2 -6599.27} C_VEL
LIN {X 0,Y 488.705,Z 508.611,A -85,B 0,C 180,E1 -6602.146,E2 -6602.146} C_VEL
LIN {X 0,Y 488.722,Z 508.609,A -85,B 0,C 180,E1 -6605.114,E2 -6605.114} C_VEL
LIN {X 0,Y 488.682,Z 508.612,A -85,B 0,C 180,E1 -6608.199,E2 -6608.199} C_VEL
LIN {X 0,Y 488.747,Z 508.605,A -85,B 0,C 180,E1 -6610.348,E2 -6610.348} C_VEL
LIN {X 0,Y 488.714,Z 508.605,A -85,B 0,C 180,E1 -6613.65,E2 -6613.65} C_VEL
LIN {X 0,Y 488.689,Z 508.611,A -85,B 0,C 180,E1 -6616.345,E2 -6616.345} C_VEL
LIN {X 0,Y 488.715,Z 508.609,A -85,B 0,C 180,E1 -6618.585,E2 -6618.585} C_VEL
LIN {X 0,Y 488.677,Z 508.609,A -85,B 0,C 180,E1 -6621.799,E2 -6621.799} C_VEL
LIN {X 0,Y 488.724,Z 508.606,A -85,B 0,C 180,E1 -6625.05,E2 -6625.05} C_VEL
LIN {X 0,Y 488.7,Z 508.607,A -85,B 0,C 180,E1 -6628.044,E2 -6628.044} C_VEL
LIN {X 0,Y 488.728,Z 508.61,A -85,B 0,C 180,E1 -6630.73,E2 -6630.73} C_VEL
LIN {X 0,Y 488.759,Z 508.6,A -85,B 0,C 180,E1 -6633.528,E2 -6633.528} C_VEL
LIN {X 0,Y 488.685,Z 508.606,A -85,B 0,C 180,E1 -6636.254,E2 -6636.254} C_VEL
LIN {X 0,Y 488.738,Z 508.604,A -85,B 0,C 180,E1 -6639.175,E2 -6639.175} C_VEL
LIN {X 0,Y 488.751,Z 508.6,A -85,B 0,C 180,E1 -6641.627,E2 -6641.627} C_VEL
LIN {X 0,Y 488.753,Z 508.606,A -85,B 0,C 180,E1 -6644.999,E2 -6644.999} C_VEL
LIN {X 0,Y 488.799,Z 508.595,A -85,B 0,C 180,E1 -6648.387,E2 -6648.387} C_VEL
LIN {X 0,Y 488.809,Z 508.593,A -85,B 0,C 180,E1 -6651.733,E2 -6651.733} C_VEL
LIN {X 0,Y 488.864,Z 508.584,A -85,B 0,C 180,E1 -6654.224,E2 -6654.224} C_VEL
LIN {X 0,Y 488.953,Z 508.576,A -85,B 0,C 180,E1 -6657.528,E2 -6657.528} C_VEL
LIN {X 0,Y 488.959,Z 508.572,A -85,B 0,C 180,E1 -6660,E2 -6660} C_VEL
LIN {X 0,Y 488.953,Z 508.577,A -85,B 0,C 180,E1 -6662.471,E2 -6662.471} C_VEL
LIN {X 0,Y 488.864,Z 508.585,A -85,B 0,C 180,E1 -6665.775,E2 -6665.775} C_VEL
LIN {X 0,Y 488.809,Z 508.593,A -85,B 0,C 180,E1 -6668.266,E2 -6668.266} C_VEL
LIN {X 0,Y 488.798,Z 508.596,A -85,B 0,C 180,E1 -6671.612,E2 -6671.612} C_VEL
LIN {X 0,Y 488.751,Z 508.607,A -85,B 0,C 180,E1 -6675,E2 -6675} C_VEL
LIN {X 0,Y 488.745,Z 508.602,A -85,B 0,C 180,E1 -6678.442,E2 -6678.442} C_VEL
LIN {X 0,Y 488.697,Z 508.614,A -85,B 0,C 180,E1 -6681.071,E2 -6681.071} C_VEL
LIN {X 0,Y 488.683,Z 508.613,A -85,B 0,C 180,E1 -6683.745,E2 -6683.745} C_VEL
LIN {X 0,Y 488.789,Z 508.604,A -85,B 0,C 180,E1 -6686.945,E2 -6686.945} C_VEL
LIN {X 0,Y 488.709,Z 508.608,A -85,B 0,C 180,E1 -6690.365,E2 -6690.365} C_VEL
LIN {X 0,Y 488.723,Z 508.612,A -85,B 0,C 180,E1 -6692.939,E2 -6692.939} C_VEL
LIN {X 0,Y 489.553,Z 514.379,A -85,B 0,C 180,E1 -6694.296,E2 -6694.296} C_VEL
LIN {X 0,Y 489.417,Z 521.266,A -85,B 0,C 180,E1 -6695.814,E2 -6695.814} C_VEL
LIN {X 0,Y 491.835,Z 532.94,A -85,B 0,C 180,E1 -6696.077,E2 -6696.077} C_VEL
LIN {X 0,Y 491.114,Z 627.507,A -85,B 0,C 180,E1 -6697.506,E2 -6697.506} C_VEL
LIN {X 0,Y 490.884,Z 640.999,A -85,B 0,C 180,E1 -6697.887,E2 -6697.887} C_VEL
LIN {X 0,Y 490.621,Z 653.503,A -85,B 0,C 180,E1 -6698.412,E2 -6698.412} C_VEL
LIN {X 0,Y 490.199,Z 665.7,A -85,B 0,C 180,E1 -6699.111,E2 -6699.111} C_VEL
LIN {X 0,Y 489.806,Z 677.243,A -85,B 0,C 180,E1 -6699.965,E2 -6699.965} C_VEL
LIN {X 0,Y 489.392,Z 687.112,A -85,B 0,C 180,E1 -6700.876,E2 -6700.876} C_VEL
LIN {X 0,Y 489.06,Z 695.404,A -85,B 0,C 180,E1 -6701.811,E2 -6701.811} C_VEL
LIN {X 0,Y 488.69,Z 703.993,A -85,B 0,C 180,E1 -6702.995,E2 -6702.995} C_VEL
LIN {X 0,Y 488.432,Z 711.214,A -85,B 0,C 180,E1 -6704.226,E2 -6704.226} C_VEL
LIN {X 0,Y 488.256,Z 717.742,A -85,B 0,C 180,E1 -6705.629,E2 -6705.629} C_VEL
LIN {X 0,Y 488.135,Z 721.997,A -85,B 0,C 180,E1 -6706.804,E2 -6706.804} C_VEL
LIN {X 0,Y 488.091,Z 723.601,A -85,B 0,C 180,E1 -6707.34,E2 -6707.34} C_VEL
LIN {X 0,Y 487.422,Z 725.43,A -85,B 0,C 180,E1 -6707.995,E2 -6707.995} C_VEL
LIN {X 0,Y 484.415,Z 727.89,A -85,B 0,C 180,E1 -6709.073,E2 -6709.073} C_VEL
LIN {X 0,Y 481.398,Z 729.545,A -85,B 0,C 180,E1 -6710.183,E2 -6710.183} C_VEL
LIN {X 0,Y 480.733,Z 730.115,A -85,B 0,C 180,E1 -6710.882,E2 -6710.882} C_VEL
LIN {X 0,Y 480.74,Z 730.49,A -85,B 0,C 180,E1 -6712.132,E2 -6712.132} C_VEL
LIN {X 0,Y 480.745,Z 729.867,A -85,B 0,C 180,E1 -6713.517,E2 -6713.517} C_VEL
LIN {X 0,Y 480.812,Z 728.094,A -85,B 0,C 180,E1 -6714.939,E2 -6714.939} C_VEL
LIN {X 0,Y 480.942,Z 725.032,A -85,B 0,C 180,E1 -6716.401,E2 -6716.401} C_VEL
LIN {X 0,Y 481.09,Z 720.45,A -85,B 0,C 180,E1 -6717.917,E2 -6717.917} C_VEL
LIN {X 0,Y 481.307,Z 714.969,A -85,B 0,C 180,E1 -6719.266,E2 -6719.266} C_VEL
LIN {X 0,Y 481.563,Z 708.751,A -85,B 0,C 180,E1 -6720.48,E2 -6720.48} C_VEL
LIN {X 0,Y 481.855,Z 700.998,A -85,B 0,C 180,E1 -6721.705,E2 -6721.705} C_VEL
LIN {X 0,Y 482.185,Z 692.855,A -85,B 0,C 180,E1 -6722.759,E2 -6722.759} C_VEL
LIN {X 0,Y 482.619,Z 683.544,A -85,B 0,C 180,E1 -6723.748,E2 -6723.748} C_VEL
LIN {X 0,Y 483.051,Z 672.643,A -85,B 0,C 180,E1 -6724.683,E2 -6724.683} C_VEL
LIN {X 0,Y 483.43,Z 662,A -85,B 0,C 180,E1 -6725.409,E2 -6725.409} C_VEL
LIN {X 0,Y 483.797,Z 649.924,A -85,B 0,C 180,E1 -6726.049,E2 -6726.049} C_VEL
LIN {X 0,Y 484.127,Z 637.035,A -85,B 0,C 180,E1 -6726.544,E2 -6726.544} C_VEL
LIN {X 0,Y 484.321,Z 624.17,A -85,B 0,C 180,E1 -6726.858,E2 -6726.858} C_VEL
LIN {X 0,Y 484.909,Z 533.045,A -85,B 0,C 180,E1 -6728.244,E2 -6728.244} C_VEL
LIN {X 0,Y 482.383,Z 520.849,A -85,B 0,C 180,E1 -6728.541,E2 -6728.541} C_VEL
LIN {X 0,Y 482.418,Z 514.446,A -85,B 0,C 180,E1 -6729.98,E2 -6729.98} C_VEL
LIN {X 0,Y 481.716,Z 509.484,A -85,B 0,C 180,E1 -6731.169,E2 -6731.169} C_VEL
LIN {X 0,Y 481.739,Z 509.481,A -85,B 0,C 180,E1 -6734.776,E2 -6734.776} C_VEL
LIN {X 0,Y 481.748,Z 509.472,A -85,B 0,C 180,E1 -6738.215,E2 -6738.215} C_VEL
LIN {X 0,Y 481.76,Z 509.47,A -85,B 0,C 180,E1 -6741.612,E2 -6741.612} C_VEL
LIN {X 0,Y 481.806,Z 509.465,A -85,B 0,C 180,E1 -6744.14,E2 -6744.14} C_VEL
LIN {X 0,Y 481.926,Z 509.451,A -85,B 0,C 180,E1 -6747.493,E2 -6747.493} C_VEL
LIN {X 0,Y 481.903,Z 509.46,A -85,B 0,C 180,E1 -6750.836,E2 -6750.836} C_VEL
LIN {X 0,Y 481.926,Z 509.452,A -85,B 0,C 180,E1 -6752.507,E2 -6752.507} C_VEL
LIN {X 0,Y 481.816,Z 509.463,A -85,B 0,C 180,E1 -6755.86,E2 -6755.86} C_VEL
LIN {X 0,Y 481.76,Z 509.471,A -85,B 0,C 180,E1 -6758.388,E2 -6758.388} C_VEL
LIN {X 0,Y 481.748,Z 509.471,A -85,B 0,C 180,E1 -6761.785,E2 -6761.785} C_VEL
LIN {X 0,Y 481.739,Z 509.477,A -85,B 0,C 180,E1 -6765.224,E2 -6765.224} C_VEL
LIN {X 0,Y 481.709,Z 509.481,A -85,B 0,C 180,E1 -6768.721,E2 -6768.721} C_VEL
LIN {X 0,Y 481.643,Z 509.487,A -85,B 0,C 180,E1 -6771.394,E2 -6771.394} C_VEL
LIN {X 0,Y 481.673,Z 509.481,A -85,B 0,C 180,E1 -6774.113,E2 -6774.113} C_VEL
LIN {X 0,Y 481.742,Z 509.479,A -85,B 0,C 180,E1 -6777.139,E2 -6777.139} C_VEL
LIN {X 0,Y 481.683,Z 509.48,A -85,B 0,C 180,E1 -6779.74,E2 -6779.74} C_VEL
LIN {X 0,Y 481.667,Z 509.485,A -85,B 0,C 180,E1 -6782.674,E2 -6782.674} C_VEL
LIN {X 0,Y 481.637,Z 509.486,A -85,B 0,C 180,E1 -6785.708,E2 -6785.708} C_VEL
LIN {X 0,Y 481.713,Z 509.48,A -85,B 0,C 180,E1 -6789.354,E2 -6789.354} C_VEL
LIN {X 0,Y 481.668,Z 509.481,A -85,B 0,C 180,E1 -6792.157,E2 -6792.157} C_VEL
LIN {X 0,Y 481.652,Z 509.485,A -85,B 0,C 180,E1 -6794.457,E2 -6794.457} C_VEL
LIN {X 0,Y 481.681,Z 509.485,A -85,B 0,C 180,E1 -6796.845,E2 -6796.845} C_VEL
LIN {X 0,Y 481.684,Z 509.479,A -85,B 0,C 180,E1 -6800.061,E2 -6800.061} C_VEL
LIN {X 0,Y 481.623,Z 509.493,A -85,B 0,C 180,E1 -6803.253,E2 -6803.253} C_VEL
LIN {X 0,Y 481.7,Z 509.478,A -85,B 0,C 180,E1 -6806.33,E2 -6806.33} C_VEL
LIN {X 0,Y 481.649,Z 509.488,A -85,B 0,C 180,E1 -6809.415,E2 -6809.415} C_VEL
LIN {X 0,Y 481.693,Z 509.478,A -85,B 0,C 180,E1 -6812.168,E2 -6812.168} C_VEL
LIN {X 0,Y 481.709,Z 509.483,A -85,B 0,C 180,E1 -6814.97,E2 -6814.97} C_VEL
LIN {X 0,Y 481.64,Z 509.486,A -85,B 0,C 180,E1 -6817.705,E2 -6817.705} C_VEL
LIN {X 0,Y 481.698,Z 509.478,A -85,B 0,C 180,E1 -6820.393,E2 -6820.393} C_VEL
LIN {X 0,Y 481.682,Z 509.487,A -85,B 0,C 180,E1 -6823.034,E2 -6823.034} C_VEL
LIN {X 0,Y 481.679,Z 509.482,A -85,B 0,C 180,E1 -6825.639,E2 -6825.639} C_VEL
LIN {X 0,Y 481.786,Z 509.466,A -85,B 0,C 180,E1 -6828.216,E2 -6828.216} C_VEL
LIN {X 0,Y 481.754,Z 509.473,A -85,B 0,C 180,E1 -6831.612,E2 -6831.612} C_VEL
LIN {X 0,Y 481.822,Z 509.462,A -85,B 0,C 180,E1 -6834.14,E2 -6834.14} C_VEL
LIN {X 0,Y 481.92,Z 509.454,A -85,B 0,C 180,E1 -6837.493,E2 -6837.493} C_VEL
LIN {X 0,Y 481.93,Z 509.449,A -85,B 0,C 180,E1 -6840,E2 -6840} C_VEL
LIN {X 0,Y 481.926,Z 509.45,A -85,B 0,C 180,E1 -6842.508,E2 -6842.508} C_VEL
LIN {X 0,Y 481.823,Z 509.463,A -85,B 0,C 180,E1 -6845.861,E2 -6845.861} C_VEL
LIN {X 0,Y 481.755,Z 509.471,A -85,B 0,C 180,E1 -6848.389,E2 -6848.389} C_VEL
LIN {X 0,Y 481.744,Z 509.474,A -85,B 0,C 180,E1 -6851.785,E2 -6851.785} C_VEL
LIN {X 0,Y 481.734,Z 509.482,A -85,B 0,C 180,E1 -6855.225,E2 -6855.225} C_VEL
LIN {X 0,Y 481.704,Z 509.479,A -85,B 0,C 180,E1 -6858.722,E2 -6858.722} C_VEL
LIN {X 0,Y 481.639,Z 509.492,A -85,B 0,C 180,E1 -6861.395,E2 -6861.395} C_VEL
LIN {X 0,Y 481.67,Z 509.481,A -85,B 0,C 180,E1 -6864.114,E2 -6864.114} C_VEL
LIN {X 0,Y 481.745,Z 509.478,A -85,B 0,C 180,E1 -6867.141,E2 -6867.141} C_VEL
LIN {X 0,Y 481.682,Z 509.482,A -85,B 0,C 180,E1 -6869.741,E2 -6869.741} C_VEL
LIN {X 0,Y 481.668,Z 509.482,A -85,B 0,C 180,E1 -6872.675,E2 -6872.675} C_VEL
LIN {X 0,Y 481.638,Z 509.488,A -85,B 0,C 180,E1 -6875.71,E2 -6875.71} C_VEL
LIN {X 0,Y 481.667,Z 509.484,A -85,B 0,C 180,E1 -6878.86,E2 -6878.86} C_VEL
LIN {X 0,Y 481.659,Z 509.484,A -85,B 0,C 180,E1 -6881.915,E2 -6881.915} C_VEL
LIN {X 0,Y 481.657,Z 509.483,A -85,B 0,C 180,E1 -6884.458,E2 -6884.458} C_VEL
LIN {X 0,Y 481.687,Z 509.481,A -85,B 0,C 180,E1 -6886.847,E2 -6886.847} C_VEL
LIN {X 0,Y 481.687,Z 509.48,A -85,B 0,C 180,E1 -6890.062,E2 -6890.062} C_VEL
LIN {X 0,Y 481.627,Z 509.493,A -85,B 0,C 180,E1 -6893.254,E2 -6893.254} C_VEL
LIN {X 0,Y 481.709,Z 509.478,A -85,B 0,C 180,E1 -6896.331,E2 -6896.331} C_VEL
LIN {X 0,Y 481.652,Z 509.492,A -85,B 0,C 180,E1 -6899.418,E2 -6899.418} C_VEL
LIN {X 0,Y 481.701,Z 509.482,A -85,B 0,C 180,E1 -6902.169,E2 -6902.169} C_VEL
LIN {X 0,Y 481.774,Z 509.624,A -85,B 0,C 180,E1 -6903.232,E2 -6903.232} C_VEL
LIN {X 0,Y 484.135,Z 521.502,A -85,B 0,C 180,E1 -6905.333,E2 -6905.333} C_VEL
LIN {X 0,Y 484.011,Z 528.734,A -85,B 0,C 180,E1 -6906.519,E2 -6906.519} C_VEL
LIN {X 0,Y 483.264,Z 546.333,A -85,B 0,C 180,E1 -6909.35,E2 -6909.35} C_VEL
LIN {X 0,Y 482.599,Z 564.244,A -85,B 0,C 180,E1 -6912.193,E2 -6912.193} C_VEL
LIN {X 0,Y 482.368,Z 572.376,A -85,B 0,C 180,E1 -6913.475,E2 -6913.475} C_VEL
LIN {X 0,Y 484.831,Z 590.548,A -85,B 0,C 180,E1 -6913.85,E2 -6913.85} C_VEL
LIN {X 0,Y 484.139,Z 681.159,A -85,B 0,C 180,E1 -6915.23,E2 -6915.23} C_VEL
LIN {X 0,Y 483.827,Z 694.432,A -85,B 0,C 180,E1 -6915.597,E2 -6915.597} C_VEL
LIN {X 0,Y 483.437,Z 707.185,A -85,B 0,C 180,E1 -6916.121,E2 -6916.121} C_VEL
LIN {X 0,Y 483.053,Z 718.539,A -85,B 0,C 180,E1 -6916.754,E2 -6916.754} C_VEL
LIN {X 0,Y 482.621,Z 730.254,A -85,B 0,C 180,E1 -6917.597,E2 -6917.597} C_VEL
LIN {X 0,Y 482.213,Z 740.799,A -85,B 0,C 180,E1 -6918.547,E2 -6918.547} C_VEL
LIN {X 0,Y 481.775,Z 749.419,A -85,B 0,C 180,E1 -6919.494,E2 -6919.494} C_VEL
LIN {X 0,Y 481.477,Z 757.378,A -85,B 0,C 180,E1 -6920.549,E2 -6920.549} C_VEL
LIN {X 0,Y 481.201,Z 765.156,A -85,B 0,C 180,E1 -6921.813,E2 -6921.813} C_VEL
LIN {X 0,Y 481.02,Z 772.317,A -85,B 0,C 180,E1 -6923.288,E2 -6923.288} C_VEL
LIN {X 0,Y 480.956,Z 777.086,A -85,B 0,C 180,E1 -6924.55,E2 -6924.55} C_VEL
LIN {X 0,Y 480.851,Z 780.726,A -85,B 0,C 180,E1 -6925.809,E2 -6925.809} C_VEL
LIN {X 0,Y 480.893,Z 782.608,A -85,B 0,C 180,E1 -6926.649,E2 -6926.649} C_VEL
LIN {X 0,Y 480.869,Z 784.015,A -85,B 0,C 180,E1 -6927.487,E2 -6927.487} C_VEL
LIN {X 0,Y 480.824,Z 785.015,A -85,B 0,C 180,E1 -6928.325,E2 -6928.325} C_VEL
LIN {X 0,Y 480.744,Z 785.832,A -85,B 0,C 180,E1 -6930,E2 -6930} C_VEL
LIN {X 0,Y 480.824,Z 784.991,A -85,B 0,C 180,E1 -6931.675,E2 -6931.675} C_VEL
LIN {X 0,Y 480.869,Z 783.979,A -85,B 0,C 180,E1 -6932.513,E2 -6932.513} C_VEL
LIN {X 0,Y 480.893,Z 782.559,A -85,B 0,C 180,E1 -6933.351,E2 -6933.351} C_VEL
LIN {X 0,Y 480.846,Z 779.574,A -85,B 0,C 180,E1 -6934.611,E2 -6934.611} C_VEL
LIN {X 0,Y 480.944,Z 775.546,A -85,B 0,C 180,E1 -6935.871,E2 -6935.871} C_VEL
LIN {X 0,Y 481.108,Z 769.351,A -85,B 0,C 180,E1 -6937.343,E2 -6937.343} C_VEL
LIN {X 0,Y 481.308,Z 762.586,A -85,B 0,C 180,E1 -6938.608,E2 -6938.608} C_VEL
LIN {X 0,Y 481.569,Z 754.197,A -85,B 0,C 180,E1 -6939.874,E2 -6939.874} C_VEL
LIN {X 0,Y 481.933,Z 745.592,A -85,B 0,C 180,E1 -6940.928,E2 -6940.928} C_VEL
LIN {X 0,Y 482.397,Z 734.987,A -85,B 0,C 180,E1 -6941.981,E2 -6941.981} C_VEL
LIN {X 0,Y 482.868,Z 723.675,A -85,B 0,C 180,E1 -6942.883,E2 -6942.883} C_VEL
LIN {X 0,Y 483.205,Z 712.925,A -85,B 0,C 180,E1 -6943.564,E2 -6943.564} C_VEL
LIN {X 0,Y 483.634,Z 701,A -85,B 0,C 180,E1 -6944.141,E2 -6944.141} C_VEL
LIN {X 0,Y 483.942,Z 687.245,A -85,B 0,C 180,E1 -6944.615,E2 -6944.615} C_VEL
LIN {X 0,Y 484.257,Z 674.86,A -85,B 0,C 180,E1 -6944.874,E2 -6944.874} C_VEL
LIN {X 0,Y 484.691,Z 588.526,A -85,B 0,C 180,E1 -6946.179,E2 -6946.179} C_VEL
LIN {X 0,Y 482.31,Z 571.835,A -85,B 0,C 180,E1 -6946.535,E2 -6946.535} C_VEL
LIN {X 0,Y 482.965,Z 552.672,A -85,B 0,C 180,E1 -6949.553,E2 -6949.553} C_VEL
LIN {X 0,Y 483.69,Z 533.312,A -85,B 0,C 180,E1 -6952.646,E2 -6952.646} C_VEL
LIN {X 0,Y 484.124,Z 522.265,A -85,B 0,C 180,E1 -6954.439,E2 -6954.439} C_VEL
LIN {X 0,Y 481.808,Z 509.724,A -85,B 0,C 180,E1 -6956.649,E2 -6956.649} C_VEL
LIN {X 0,Y 481.749,Z 509.479,A -85,B 0,C 180,E1 -6956.887,E2 -6956.887} C_VEL
LIN {X 0,Y 481.679,Z 509.484,A -85,B 0,C 180,E1 -6959.74,E2 -6959.74} C_VEL
LIN {X 0,Y 481.673,Z 509.488,A -85,B 0,C 180,E1 -6962.673,E2 -6962.673} C_VEL
LIN {X 0,Y 481.642,Z 509.488,A -85,B 0,C 180,E1 -6965.708,E2 -6965.708} C_VEL
LIN {X 0,Y 481.713,Z 509.478,A -85,B 0,C 180,E1 -6969.353,E2 -6969.353} C_VEL
LIN {X 0,Y 481.672,Z 509.484,A -85,B 0,C 180,E1 -6972.157,E2 -6972.157} C_VEL
LIN {X 0,Y 481.657,Z 509.489,A -85,B 0,C 180,E1 -6974.456,E2 -6974.456} C_VEL
LIN {X 0,Y 481.65,Z 509.483,A -85,B 0,C 180,E1 -6977.839,E2 -6977.839} C_VEL
LIN {X 0,Y 481.676,Z 509.486,A -85,B 0,C 180,E1 -6980.65,E2 -6980.65} C_VEL
LIN {X 0,Y 481.628,Z 509.488,A -85,B 0,C 180,E1 -6983.374,E2 -6983.374} C_VEL
LIN {X 0,Y 481.704,Z 509.478,A -85,B 0,C 180,E1 -6986.329,E2 -6986.329} C_VEL
LIN {X 0,Y 481.652,Z 509.485,A -85,B 0,C 180,E1 -6989.415,E2 -6989.415} C_VEL
LIN {X 0,Y 481.696,Z 509.478,A -85,B 0,C 180,E1 -6992.167,E2 -6992.167} C_VEL
LIN {X 0,Y 481.711,Z 509.48,A -85,B 0,C 180,E1 -6994.969,E2 -6994.969} C_VEL
LIN {X 0,Y 481.642,Z 509.485,A -85,B 0,C 180,E1 -6997.704,E2 -6997.704} C_VEL
LIN {X 0,Y 481.701,Z 509.479,A -85,B 0,C 180,E1 -7000.392,E2 -7000.392} C_VEL
LIN {X 0,Y 481.684,Z 509.485,A -85,B 0,C 180,E1 -7003.033,E2 -7003.033} C_VEL
LIN {X 0,Y 481.682,Z 509.48,A -85,B 0,C 180,E1 -7005.638,E2 -7005.638} C_VEL
LIN {X 0,Y 481.744,Z 509.473,A -85,B 0,C 180,E1 -7008.215,E2 -7008.215} C_VEL
LIN {X 0,Y 481.755,Z 509.472,A -85,B 0,C 180,E1 -7011.611,E2 -7011.611} C_VEL
LIN {X 0,Y 481.822,Z 509.461,A -85,B 0,C 180,E1 -7014.139,E2 -7014.139} C_VEL
LIN {X 0,Y 481.92,Z 509.452,A -85,B 0,C 180,E1 -7017.492,E2 -7017.492} C_VEL
LIN {X 0,Y 481.93,Z 509.448,A -85,B 0,C 180,E1 -7020,E2 -7020} C_VEL
LIN {X 0,Y 481.92,Z 509.453,A -85,B 0,C 180,E1 -7022.507,E2 -7022.507} C_VEL
LIN {X 0,Y 481.822,Z 509.462,A -85,B 0,C 180,E1 -7025.86,E2 -7025.86} C_VEL
LIN {X 0,Y 481.754,Z 509.473,A -85,B 0,C 180,E1 -7028.388,E2 -7028.388} C_VEL
LIN {X 0,Y 481.742,Z 509.474,A -85,B 0,C 180,E1 -7031.785,E2 -7031.785} C_VEL
LIN {X 0,Y 481.732,Z 509.481,A -85,B 0,C 180,E1 -7035.224,E2 -7035.224} C_VEL
LIN {X 0,Y 481.702,Z 509.482,A -85,B 0,C 180,E1 -7038.722,E2 -7038.722} C_VEL
LIN {X 0,Y 481.637,Z 509.493,A -85,B 0,C 180,E1 -7041.395,E2 -7041.395} C_VEL
LIN {X 0,Y 481.667,Z 509.486,A -85,B 0,C 180,E1 -7044.113,E2 -7044.113} C_VEL
LIN {X 0,Y 481.742,Z 509.482,A -85,B 0,C 180,E1 -7047.141,E2 -7047.141} C_VEL
LIN {X 0,Y 481.679,Z 509.486,A -85,B 0,C 180,E1 -7049.741,E2 -7049.741} C_VEL
LIN {X 0,Y 481.723,Z 509.622,A -85,B 0,C 180,E1 -7052.794,E2 -7052.794} C_VEL
LIN {X 0,Y 482.586,Z 515.422,A -85,B 0,C 180,E1 -7054.178,E2 -7054.178} C_VEL
LIN {X 0,Y 482.455,Z 521.463,A -85,B 0,C 180,E1 -7055.561,E2 -7055.561} C_VEL
LIN {X 0,Y 484.966,Z 533.253,A -85,B 0,C 180,E1 -7055.842,E2 -7055.842} C_VEL
LIN {X 0,Y 484.274,Z 627.438,A -85,B 0,C 180,E1 -7057.287,E2 -7057.287} C_VEL
LIN {X 0,Y 484.03,Z 641.006,A -85,B 0,C 180,E1 -7057.67,E2 -7057.67} C_VEL
LIN {X 0,Y 483.78,Z 652.805,A -85,B 0,C 180,E1 -7058.164,E2 -7058.164} C_VEL
LIN {X 0,Y 483.367,Z 664.691,A -85,B 0,C 180,E1 -7058.83,E2 -7058.83} C_VEL
LIN {X 0,Y 482.973,Z 675.862,A -85,B 0,C 180,E1 -7059.644,E2 -7059.644} C_VEL
LIN {X 0,Y 482.526,Z 686.07,A -85,B 0,C 180,E1 -7060.571,E2 -7060.571} C_VEL
LIN {X 0,Y 482.119,Z 694.877,A -85,B 0,C 180,E1 -7061.549,E2 -7061.549} C_VEL
LIN {X 0,Y 481.778,Z 702.93,A -85,B 0,C 180,E1 -7062.636,E2 -7062.636} C_VEL
LIN {X 0,Y 481.491,Z 710.076,A -85,B 0,C 180,E1 -7063.819,E2 -7063.819} C_VEL
LIN {X 0,Y 481.223,Z 716.916,A -85,B 0,C 180,E1 -7065.241,E2 -7065.241} C_VEL
LIN {X 0,Y 481.076,Z 722.111,A -85,B 0,C 180,E1 -7066.638,E2 -7066.638} C_VEL
LIN {X 0,Y 480.971,Z 725.307,A -85,B 0,C 180,E1 -7067.768,E2 -7067.768} C_VEL
LIN {X 0,Y 480.791,Z 728.655,A -85,B 0,C 180,E1 -7069.473,E2 -7069.473} C_VEL
LIN {X 0,Y 480.733,Z 730.115,A -85,B 0,C 180,E1 -7070.882,E2 -7070.882} C_VEL
LIN {X 0,Y 480.097,Z 730.468,A -85,B 0,C 180,E1 -7071.581,E2 -7071.581} C_VEL
LIN {X 0,Y 477.21,Z 730.572,A -85,B 0,C 180,E1 -7072.717,E2 -7072.717} C_VEL
LIN {X 0,Y 474.768,Z 730.118,A -85,B 0,C 180,E1 -7073.631,E2 -7073.631} C_VEL
LIN {X 0,Y 473.751,Z 729.427,A -85,B 0,C 180,E1 -7074.334,E2 -7074.334} C_VEL
LIN {X 0,Y 473.686,Z 729.103,A -85,B 0,C 180,E1 -7074.572,E2 -7074.572} C_VEL
LIN {X 0,Y 473.838,Z 726.192,A -85,B 0,C 180,E1 -7076.159,E2 -7076.159} C_VEL
LIN {X 0,Y 473.978,Z 721.728,A -85,B 0,C 180,E1 -7077.739,E2 -7077.739} C_VEL
LIN {X 0,Y 474.24,Z 715.855,A -85,B 0,C 180,E1 -7079.263,E2 -7079.263} C_VEL
LIN {X 0,Y 474.506,Z 709.74,A -85,B 0,C 180,E1 -7080.498,E2 -7080.498} C_VEL
LIN {X 0,Y 474.832,Z 702.175,A -85,B 0,C 180,E1 -7081.73,E2 -7081.73} C_VEL
LIN {X 0,Y 475.238,Z 692.91,A -85,B 0,C 180,E1 -7082.952,E2 -7082.952} C_VEL
LIN {X 0,Y 475.718,Z 682.701,A -85,B 0,C 180,E1 -7084.035,E2 -7084.035} C_VEL
LIN {X 0,Y 476.143,Z 672.669,A -85,B 0,C 180,E1 -7084.891,E2 -7084.891} C_VEL
LIN {X 0,Y 476.58,Z 661.1,A -85,B 0,C 180,E1 -7085.678,E2 -7085.678} C_VEL
LIN {X 0,Y 476.995,Z 648.527,A -85,B 0,C 180,E1 -7086.331,E2 -7086.331} C_VEL
LIN {X 0,Y 477.281,Z 635.62,A -85,B 0,C 180,E1 -7086.803,E2 -7086.803} C_VEL
LIN {X 0,Y 477.486,Z 622.824,A -85,B 0,C 180,E1 -7087.1,E2 -7087.1} C_VEL
LIN {X 0,Y 478.118,Z 534.047,A -85,B 0,C 180,E1 -7088.468,E2 -7088.468} C_VEL
LIN {X 0,Y 475.43,Z 521.168,A -85,B 0,C 180,E1 -7088.794,E2 -7088.794} C_VEL
LIN {X 0,Y 475.436,Z 515.337,A -85,B 0,C 180,E1 -7090.124,E2 -7090.124} C_VEL
LIN {X 0,Y 474.687,Z 510.359,A -85,B 0,C 180,E1 -7091.36,E2 -7091.36} C_VEL
LIN {X 0,Y 474.696,Z 510.356,A -85,B 0,C 180,E1 -7094.545,E2 -7094.545} C_VEL
LIN {X 0,Y 474.701,Z 510.349,A -85,B 0,C 180,E1 -7098.038,E2 -7098.038} C_VEL
LIN {X 0,Y 474.725,Z 510.348,A -85,B 0,C 180,E1 -7101.487,E2 -7101.487} C_VEL
LIN {X 0,Y 474.768,Z 510.341,A -85,B 0,C 180,E1 -7104.052,E2 -7104.052} C_VEL
LIN {X 0,Y 474.892,Z 510.327,A -85,B 0,C 180,E1 -7107.455,E2 -7107.455} C_VEL
LIN {X 0,Y 474.91,Z 510.323,A -85,B 0,C 180,E1 -7110,E2 -7110} C_VEL
LIN {X 0,Y 474.892,Z 510.329,A -85,B 0,C 180,E1 -7112.545,E2 -7112.545} C_VEL
LIN {X 0,Y 474.778,Z 510.339,A -85,B 0,C 180,E1 -7115.947,E2 -7115.947} C_VEL
LIN {X 0,Y 474.725,Z 510.349,A -85,B 0,C 180,E1 -7118.513,E2 -7118.513} C_VEL
LIN {X 0,Y 474.701,Z 510.349,A -85,B 0,C 180,E1 -7121.962,E2 -7121.962} C_VEL
LIN {X 0,Y 474.696,Z 510.352,A -85,B 0,C 180,E1 -7125.455,E2 -7125.455} C_VEL
LIN {X 0,Y 474.662,Z 510.362,A -85,B 0,C 180,E1 -7129.01,E2 -7129.01} C_VEL
LIN {X 0,Y 474.586,Z 510.364,A -85,B 0,C 180,E1 -7131.728,E2 -7131.728} C_VEL
LIN {X 0,Y 474.654,Z 510.357,A -85,B 0,C 180,E1 -7134.492,E2 -7134.492} C_VEL
LIN {X 0,Y 474.694,Z 510.354,A -85,B 0,C 180,E1 -7137.338,E2 -7137.338} C_VEL
LIN {X 0,Y 474.612,Z 510.366,A -85,B 0,C 180,E1 -7140.813,E2 -7140.813} C_VEL
LIN {X 0,Y 474.632,Z 510.358,A -85,B 0,C 180,E1 -7143.984,E2 -7143.984} C_VEL
LIN {X 0,Y 474.572,Z 510.372,A -85,B 0,C 180,E1 -7146.9,E2 -7146.9} C_VEL
LIN {X 0,Y 474.648,Z 510.357,A -85,B 0,C 180,E1 -7149.651,E2 -7149.651} C_VEL
LIN {X 0,Y 474.645,Z 510.363,A -85,B 0,C 180,E1 -7152.93,E2 -7152.93} C_VEL
LIN {X 0,Y 474.61,Z 510.361,A -85,B 0,C 180,E1 -7155.896,E2 -7155.896} C_VEL
LIN {X 0,Y 474.637,Z 510.366,A -85,B 0,C 180,E1 -7159.038,E2 -7159.038} C_VEL
LIN {X 0,Y 474.612,Z 510.362,A -85,B 0,C 180,E1 -7161.702,E2 -7161.702} C_VEL
LIN {X 0,Y 474.622,Z 510.363,A -85,B 0,C 180,E1 -7164.726,E2 -7164.726} C_VEL
LIN {X 0,Y 474.628,Z 510.359,A -85,B 0,C 180,E1 -7167.788,E2 -7167.788} C_VEL
LIN {X 0,Y 474.623,Z 510.364,A -85,B 0,C 180,E1 -7170.882,E2 -7170.882} C_VEL
LIN {X 0,Y 474.657,Z 510.357,A -85,B 0,C 180,E1 -7173.629,E2 -7173.629} C_VEL
LIN {X 0,Y 474.625,Z 510.361,A -85,B 0,C 180,E1 -7176.641,E2 -7176.641} C_VEL
LIN {X 0,Y 474.646,Z 510.356,A -85,B 0,C 180,E1 -7180.09,E2 -7180.09} C_VEL
LIN {X 0,Y 474.641,Z 510.36,A -85,B 0,C 180,E1 -7182.775,E2 -7182.775} C_VEL
LIN {X 0,Y 474.638,Z 510.362,A -85,B 0,C 180,E1 -7185.421,E2 -7185.421} C_VEL
LIN {X 0,Y 474.73,Z 510.346,A -85,B 0,C 180,E1 -7188.039,E2 -7188.039} C_VEL
LIN {X 0,Y 474.72,Z 510.351,A -85,B 0,C 180,E1 -7191.487,E2 -7191.487} C_VEL
LIN {X 0,Y 474.782,Z 510.339,A -85,B 0,C 180,E1 -7194.053,E2 -7194.053} C_VEL
LIN {X 0,Y 474.886,Z 510.331,A -85,B 0,C 180,E1 -7197.456,E2 -7197.456} C_VEL
LIN {X 0,Y 474.868,Z 510.332,A -85,B 0,C 180,E1 -7200.848,E2 -7200.848} C_VEL
LIN {X 0,Y 474.892,Z 510.326,A -85,B 0,C 180,E1 -7202.545,E2 -7202.545} C_VEL
LIN {X 0,Y 474.783,Z 510.34,A -85,B 0,C 180,E1 -7205.948,E2 -7205.948} C_VEL
LIN {X 0,Y 474.72,Z 510.347,A -85,B 0,C 180,E1 -7208.514,E2 -7208.514} C_VEL
LIN {X 0,Y 474.697,Z 510.35,A -85,B 0,C 180,E1 -7211.963,E2 -7211.963} C_VEL
LIN {X 0,Y 474.691,Z 510.356,A -85,B 0,C 180,E1 -7215.456,E2 -7215.456} C_VEL
LIN {X 0,Y 474.658,Z 510.359,A -85,B 0,C 180,E1 -7219.011,E2 -7219.011} C_VEL
LIN {X 0,Y 474.583,Z 510.366,A -85,B 0,C 180,E1 -7221.73,E2 -7221.73} C_VEL
LIN {X 0,Y 474.652,Z 510.356,A -85,B 0,C 180,E1 -7224.494,E2 -7224.494} C_VEL
LIN {X 0,Y 474.692,Z 510.358,A -85,B 0,C 180,E1 -7227.34,E2 -7227.34} C_VEL
LIN {X 0,Y 474.611,Z 510.363,A -85,B 0,C 180,E1 -7230.814,E2 -7230.814} C_VEL
LIN {X 0,Y 474.633,Z 510.359,A -85,B 0,C 180,E1 -7233.985,E2 -7233.985} C_VEL
LIN {X 0,Y 474.572,Z 510.368,A -85,B 0,C 180,E1 -7236.901,E2 -7236.901} C_VEL
LIN {X 0,Y 474.623,Z 510.363,A -85,B 0,C 180,E1 -7239.649,E2 -7239.649} C_VEL
LIN {X 0,Y 474.632,Z 510.361,A -85,B 0,C 180,E1 -7242.933,E2 -7242.933} C_VEL
LIN {X 0,Y 474.615,Z 510.362,A -85,B 0,C 180,E1 -7245.897,E2 -7245.897} C_VEL
LIN {X 0,Y 474.643,Z 510.36,A -85,B 0,C 180,E1 -7249.039,E2 -7249.039} C_VEL
LIN {X 0,Y 474.615,Z 510.364,A -85,B 0,C 180,E1 -7251.704,E2 -7251.704} C_VEL
LIN {X 0,Y 474.628,Z 510.359,A -85,B 0,C 180,E1 -7254.727,E2 -7254.727} C_VEL
LIN {X 0,Y 474.637,Z 510.363,A -85,B 0,C 180,E1 -7257.789,E2 -7257.789} C_VEL
LIN {X 0,Y 474.625,Z 510.364,A -85,B 0,C 180,E1 -7260.885,E2 -7260.885} C_VEL
LIN {X 0,Y 474.727,Z 510.472,A -85,B 0,C 180,E1 -7263.01,E2 -7263.01} C_VEL
LIN {X 0,Y 477.323,Z 523.916,A -85,B 0,C 180,E1 -7265.422,E2 -7265.422} C_VEL
LIN {X 0,Y 476.481,Z 543.212,A -85,B 0,C 180,E1 -7268.589,E2 -7268.589} C_VEL
LIN {X 0,Y 475.755,Z 561.111,A -85,B 0,C 180,E1 -7271.482,E2 -7271.482} C_VEL
LIN {X 0,Y 475.362,Z 572.002,A -85,B 0,C 180,E1 -7273.226,E2 -7273.226} C_VEL
LIN {X 0,Y 478.015,Z 591.045,A -85,B 0,C 180,E1 -7273.628,E2 -7273.628} C_VEL
LIN {X 0,Y 477.28,Z 680.525,A -85,B 0,C 180,E1 -7275.013,E2 -7275.013} C_VEL
LIN {X 0,Y 476.952,Z 693.885,A -85,B 0,C 180,E1 -7275.384,E2 -7275.384} C_VEL
LIN {X 0,Y 476.531,Z 706.679,A -85,B 0,C 180,E1 -7275.916,E2 -7275.916} C_VEL
LIN {X 0,Y 476.101,Z 718.066,A -85,B 0,C 180,E1 -7276.557,E2 -7276.557} C_VEL
LIN {X 0,Y 475.666,Z 729.153,A -85,B 0,C 180,E1 -7277.359,E2 -7277.359} C_VEL
LIN {X 0,Y 475.27,Z 739.284,A -85,B 0,C 180,E1 -7278.269,E2 -7278.269} C_VEL
LIN {X 0,Y 474.755,Z 748.99,A -85,B 0,C 180,E1 -7279.337,E2 -7279.337} C_VEL
LIN {X 0,Y 474.445,Z 756.955,A -85,B 0,C 180,E1 -7280.407,E2 -7280.407} C_VEL
LIN {X 0,Y 474.153,Z 764.74,A -85,B 0,C 180,E1 -7281.691,E2 -7281.691} C_VEL
LIN {X 0,Y 473.936,Z 771.904,A -85,B 0,C 180,E1 -7283.187,E2 -7283.187} C_VEL
LIN {X 0,Y 473.867,Z 776.676,A -85,B 0,C 180,E1 -7284.468,E2 -7284.468} C_VEL
LIN {X 0,Y 473.754,Z 780.317,A -85,B 0,C 180,E1 -7285.746,E2 -7285.746} C_VEL
LIN {X 0,Y 473.819,Z 782.202,A -85,B 0,C 180,E1 -7286.599,E2 -7286.599} C_VEL
LIN {X 0,Y 473.783,Z 783.609,A -85,B 0,C 180,E1 -7287.449,E2 -7287.449} C_VEL
LIN {X 0,Y 473.758,Z 784.609,A -85,B 0,C 180,E1 -7288.3,E2 -7288.3} C_VEL
LIN {X 0,Y 473.67,Z 785.425,A -85,B 0,C 180,E1 -7290,E2 -7290} C_VEL
LIN {X 0,Y 473.758,Z 784.58,A -85,B 0,C 180,E1 -7291.7,E2 -7291.7} C_VEL
LIN {X 0,Y 473.783,Z 783.565,A -85,B 0,C 180,E1 -7292.551,E2 -7292.551} C_VEL
LIN {X 0,Y 473.819,Z 782.144,A -85,B 0,C 180,E1 -7293.401,E2 -7293.401} C_VEL
LIN {X 0,Y 473.769,Z 779.154,A -85,B 0,C 180,E1 -7294.68,E2 -7294.68} C_VEL
LIN {X 0,Y 473.85,Z 775.118,A -85,B 0,C 180,E1 -7295.959,E2 -7295.959} C_VEL
LIN {X 0,Y 474.017,Z 768.913,A -85,B 0,C 180,E1 -7297.454,E2 -7297.454} C_VEL
LIN {X 0,Y 474.22,Z 762.141,A -85,B 0,C 180,E1 -7298.737,E2 -7298.737} C_VEL
LIN {X 0,Y 474.512,Z 753.747,A -85,B 0,C 180,E1 -7300.022,E2 -7300.022} C_VEL
LIN {X 0,Y 474.909,Z 745.136,A -85,B 0,C 180,E1 -7301.092,E2 -7301.092} C_VEL
LIN {X 0,Y 475.36,Z 734.774,A -85,B 0,C 180,E1 -7302.138,E2 -7302.138} C_VEL
LIN {X 0,Y 475.871,Z 724.289,A -85,B 0,C 180,E1 -7302.994,E2 -7302.994} C_VEL
LIN {X 0,Y 476.276,Z 712.447,A -85,B 0,C 180,E1 -7303.765,E2 -7303.765} C_VEL
LIN {X 0,Y 476.745,Z 699.198,A -85,B 0,C 180,E1 -7304.404,E2 -7304.404} C_VEL
LIN {X 0,Y 477.118,Z 685.813,A -85,B 0,C 180,E1 -7304.856,E2 -7304.856} C_VEL
LIN {X 0,Y 477.4,Z 672.511,A -85,B 0,C 180,E1 -7305.12,E2 -7305.12} C_VEL
LIN {X 0,Y 477.845,Z 589.269,A -85,B 0,C 180,E1 -7306.4,E2 -7306.4} C_VEL
LIN {X 0,Y 475.336,Z 571.412,A -85,B 0,C 180,E1 -7306.785,E2 -7306.785} C_VEL
LIN {X 0,Y 475.983,Z 552.266,A -85,B 0,C 180,E1 -7309.852,E2 -7309.852} C_VEL
LIN {X 0,Y 476.746,Z 534.33,A -85,B 0,C 180,E1 -7312.765,E2 -7312.765} C_VEL
LIN {X 0,Y 477.184,Z 523.298,A -85,B 0,C 180,E1 -7314.586,E2 -7314.586} C_VEL
LIN {X 0,Y 474.717,Z 510.355,A -85,B 0,C 180,E1 -7316.931,E2 -7316.931} C_VEL
LIN {X 0,Y 474.606,Z 510.368,A -85,B 0,C 180,E1 -7320.229,E2 -7320.229} C_VEL
LIN {X 0,Y 474.643,Z 510.363,A -85,B 0,C 180,E1 -7323.219,E2 -7323.219} C_VEL
LIN {X 0,Y 474.592,Z 510.37,A -85,B 0,C 180,E1 -7326.322,E2 -7326.322} C_VEL
LIN {X 0,Y 474.649,Z 510.357,A -85,B 0,C 180,E1 -7329.65,E2 -7329.65} C_VEL
LIN {X 0,Y 474.65,Z 510.362,A -85,B 0,C 180,E1 -7332.929,E2 -7332.929} C_VEL
LIN {X 0,Y 474.612,Z 510.361,A -85,B 0,C 180,E1 -7335.895,E2 -7335.895} C_VEL
LIN {X 0,Y 474.628,Z 510.363,A -85,B 0,C 180,E1 -7339.039,E2 -7339.039} C_VEL
LIN {X 0,Y 474.607,Z 510.362,A -85,B 0,C 180,E1 -7341.703,E2 -7341.703} C_VEL
LIN {X 0,Y 474.626,Z 510.367,A -85,B 0,C 180,E1 -7344.725,E2 -7344.725} C_VEL
LIN {X 0,Y 474.632,Z 510.359,A -85,B 0,C 180,E1 -7347.787,E2 -7347.787} C_VEL
LIN {X 0,Y 474.626,Z 510.366,A -85,B 0,C 180,E1 -7350.882,E2 -7350.882} C_VEL
LIN {X 0,Y 474.659,Z 510.356,A -85,B 0,C 180,E1 -7353.628,E2 -7353.628} C_VEL
LIN {X 0,Y 474.628,Z 510.361,A -85,B 0,C 180,E1 -7356.64,E2 -7356.64} C_VEL
LIN {X 0,Y 474.649,Z 510.355,A -85,B 0,C 180,E1 -7360.089,E2 -7360.089} C_VEL
LIN {X 0,Y 474.643,Z 510.361,A -85,B 0,C 180,E1 -7362.774,E2 -7362.774} C_VEL
LIN {X 0,Y 474.64,Z 510.358,A -85,B 0,C 180,E1 -7365.42,E2 -7365.42} C_VEL
LIN {X 0,Y 474.697,Z 510.35,A -85,B 0,C 180,E1 -7368.037,E2 -7368.037} C_VEL
LIN {X 0,Y 474.72,Z 510.35,A -85,B 0,C 180,E1 -7371.486,E2 -7371.486} C_VEL
LIN {X 0,Y 474.782,Z 510.337,A -85,B 0,C 180,E1 -7374.052,E2 -7374.052} C_VEL
LIN {X 0,Y 474.886,Z 510.329,A -85,B 0,C 180,E1 -7377.455,E2 -7377.455} C_VEL
LIN {X 0,Y 474.868,Z 510.333,A -85,B 0,C 180,E1 -7380.848,E2 -7380.848} C_VEL
LIN {X 0,Y 474.886,Z 510.33,A -85,B 0,C 180,E1 -7382.544,E2 -7382.544} C_VEL
LIN {X 0,Y 474.782,Z 510.339,A -85,B 0,C 180,E1 -7385.947,E2 -7385.947} C_VEL
LIN {X 0,Y 474.719,Z 510.35,A -85,B 0,C 180,E1 -7388.513,E2 -7388.513} C_VEL
LIN {X 0,Y 474.695,Z 510.351,A -85,B 0,C 180,E1 -7391.962,E2 -7391.962} C_VEL
LIN {X 0,Y 474.689,Z 510.356,A -85,B 0,C 180,E1 -7395.456,E2 -7395.456} C_VEL
LIN {X 0,Y 474.656,Z 510.363,A -85,B 0,C 180,E1 -7399.01,E2 -7399.01} C_VEL
LIN {X 0,Y 474.58,Z 510.369,A -85,B 0,C 180,E1 -7401.729,E2 -7401.729} C_VEL
LIN {X 0,Y 474.649,Z 510.361,A -85,B 0,C 180,E1 -7404.493,E2 -7404.493} C_VEL
LIN {X 0,Y 474.689,Z 510.361,A -85,B 0,C 180,E1 -7407.339,E2 -7407.339} C_VEL
LIN {X 0,Y 474.601,Z 510.369,A -85,B 0,C 180,E1 -7410.812,E2 -7410.812} C_VEL
LIN {X 0,Y 474.659,Z 510.389,A -85,B 0,C 180,E1 -7412.573,E2 -7412.573} C_VEL
LIN {X 0,Y 475.637,Z 516.933,A -85,B 0,C 180,E1 -7414.164,E2 -7414.164} C_VEL
LIN {X 0,Y 475.518,Z 521.943,A -85,B 0,C 180,E1 -7415.319,E2 -7415.319} C_VEL
LIN {X 0,Y 478.22,Z 534.838,A -85,B 0,C 180,E1 -7415.625,E2 -7415.625} C_VEL
LIN {X 0,Y 477.426,Z 628.451,A -85,B 0,C 180,E1 -7417.087,E2 -7417.087} C_VEL
LIN {X 0,Y 477.136,Z 642.428,A -85,B 0,C 180,E1 -7417.497,E2 -7417.497} C_VEL
LIN {X 0,Y 476.821,Z 655.279,A -85,B 0,C 180,E1 -7418.065,E2 -7418.065} C_VEL
LIN {X 0,Y 476.363,Z 667.925,A -85,B 0,C 180,E1 -7418.829,E2 -7418.829} C_VEL
LIN {X 0,Y 475.948,Z 678.132,A -85,B 0,C 180,E1 -7419.617,E2 -7419.617} C_VEL
LIN {X 0,Y 475.481,Z 688.113,A -85,B 0,C 180,E1 -7420.568,E2 -7420.568} C_VEL
LIN {X 0,Y 475.037,Z 697.962,A -85,B 0,C 180,E1 -7421.74,E2 -7421.74} C_VEL
LIN {X 0,Y 474.641,Z 706.083,A -85,B 0,C 180,E1 -7422.931,E2 -7422.931} C_VEL
LIN {X 0,Y 474.309,Z 714.003,A -85,B 0,C 180,E1 -7424.393,E2 -7424.393} C_VEL
LIN {X 0,Y 474.115,Z 720.06,A -85,B 0,C 180,E1 -7425.839,E2 -7425.839} C_VEL
LIN {X 0,Y 473.976,Z 723.833,A -85,B 0,C 180,E1 -7426.995,E2 -7426.995} C_VEL
LIN {X 0,Y 473.852,Z 726.719,A -85,B 0,C 180,E1 -7428.133,E2 -7428.133} C_VEL
LIN {X 0,Y 473.74,Z 728.801,A -85,B 0,C 180,E1 -7429.252,E2 -7429.252} C_VEL
LIN {X 0,Y 473.635,Z 730.477,A -85,B 0,C 180,E1 -7430.879,E2 -7430.879} C_VEL
LIN {X 0,Y 473.642,Z 730.881,A -85,B 0,C 180,E1 -7431.852,E2 -7431.852} C_VEL
LIN {X 0,Y 473.662,Z 730.484,A -85,B 0,C 180,E1 -7433.247,E2 -7433.247} C_VEL
LIN {X 0,Y 473.686,Z 729.103,A -85,B 0,C 180,E1 -7434.572,E2 -7434.572} C_VEL
LIN {X 0,Y 473.073,Z 728.145,A -85,B 0,C 180,E1 -7435.274,E2 -7435.274} C_VEL
LIN {X 0,Y 470.283,Z 725.961,A -85,B 0,C 180,E1 -7436.4,E2 -7436.4} C_VEL
LIN {X 0,Y 467.955,Z 723.686,A -85,B 0,C 180,E1 -7437.29,E2 -7437.29} C_VEL
LIN {X 0,Y 467.031,Z 721.647,A -85,B 0,C 180,E1 -7437.965,E2 -7437.965} C_VEL
LIN {X 0,Y 466.999,Z 720.883,A -85,B 0,C 180,E1 -7438.19,E2 -7438.19} C_VEL
LIN {X 0,Y 467.285,Z 714.512,A -85,B 0,C 180,E1 -7439.746,E2 -7439.746} C_VEL
LIN {X 0,Y 467.587,Z 708.166,A -85,B 0,C 180,E1 -7440.968,E2 -7440.968} C_VEL
LIN {X 0,Y 467.988,Z 699.927,A -85,B 0,C 180,E1 -7442.255,E2 -7442.255} C_VEL
LIN {X 0,Y 468.483,Z 690.028,A -85,B 0,C 180,E1 -7443.486,E2 -7443.486} C_VEL
LIN {X 0,Y 468.921,Z 680.198,A -85,B 0,C 180,E1 -7444.476,E2 -7444.476} C_VEL
LIN {X 0,Y 469.398,Z 669.981,A -85,B 0,C 180,E1 -7445.31,E2 -7445.31} C_VEL
LIN {X 0,Y 469.782,Z 657.915,A -85,B 0,C 180,E1 -7446.085,E2 -7446.085} C_VEL
LIN {X 0,Y 470.184,Z 645.878,A -85,B 0,C 180,E1 -7446.666,E2 -7446.666} C_VEL
LIN {X 0,Y 470.471,Z 632.624,A -85,B 0,C 180,E1 -7447.117,E2 -7447.117} C_VEL
LIN {X 0,Y 470.676,Z 617.071,A -85,B 0,C 180,E1 -7447.417,E2 -7447.417} C_VEL
LIN {X 0,Y 471.392,Z 535.413,A -85,B 0,C 180,E1 -7448.69,E2 -7448.69} C_VEL
LIN {X 0,Y 468.456,Z 521.541,A -85,B 0,C 180,E1 -7449.041,E2 -7449.041} C_VEL
LIN {X 0,Y 468.43,Z 516.231,A -85,B 0,C 180,E1 -7450.271,E2 -7450.271} C_VEL
LIN {X 0,Y 467.632,Z 511.237,A -85,B 0,C 180,E1 -7451.505,E2 -7451.505} C_VEL
LIN {X 0,Y 467.635,Z 511.233,A -85,B 0,C 180,E1 -7454.305,E2 -7454.305} C_VEL
LIN {X 0,Y 467.653,Z 511.227,A -85,B 0,C 180,E1 -7457.855,E2 -7457.855} C_VEL
LIN {X 0,Y 467.679,Z 511.226,A -85,B 0,C 180,E1 -7461.357,E2 -7461.357} C_VEL
LIN {X 0,Y 467.732,Z 511.217,A -85,B 0,C 180,E1 -7463.963,E2 -7463.963} C_VEL
LIN {X 0,Y 467.858,Z 511.204,A -85,B 0,C 180,E1 -7467.417,E2 -7467.417} C_VEL
LIN {X 0,Y 467.88,Z 511.199,A -85,B 0,C 180,E1 -7470,E2 -7470} C_VEL
LIN {X 0,Y 467.858,Z 511.205,A -85,B 0,C 180,E1 -7472.583,E2 -7472.583} C_VEL
LIN {X 0,Y 467.743,Z 511.216,A -85,B 0,C 180,E1 -7476.037,E2 -7476.037} C_VEL
LIN {X 0,Y 467.679,Z 511.228,A -85,B 0,C 180,E1 -7478.643,E2 -7478.643} C_VEL
LIN {X 0,Y 467.653,Z 511.227,A -85,B 0,C 180,E1 -7482.145,E2 -7482.145} C_VEL
LIN {X 0,Y 467.635,Z 511.23,A -85,B 0,C 180,E1 -7485.695,E2 -7485.695} C_VEL
LIN {X 0,Y 467.614,Z 511.237,A -85,B 0,C 180,E1 -7488.765,E2 -7488.765} C_VEL
LIN {X 0,Y 467.577,Z 511.241,A -85,B 0,C 180,E1 -7491.268,E2 -7491.268} C_VEL
LIN {X 0,Y 467.568,Z 511.238,A -85,B 0,C 180,E1 -7493.943,E2 -7493.943} C_VEL
LIN {X 0,Y 467.612,Z 511.238,A -85,B 0,C 180,E1 -7496.8,E2 -7496.8} C_VEL
LIN {X 0,Y 467.584,Z 511.236,A -85,B 0,C 180,E1 -7499.735,E2 -7499.735} C_VEL
LIN {X 0,Y 467.578,Z 511.241,A -85,B 0,C 180,E1 -7502.758,E2 -7502.758} C_VEL
LIN {X 0,Y 467.551,Z 511.24,A -85,B 0,C 180,E1 -7505.889,E2 -7505.889} C_VEL
LIN {X 0,Y 467.612,Z 511.239,A -85,B 0,C 180,E1 -7509.141,E2 -7509.141} C_VEL
LIN {X 0,Y 467.612,Z 511.235,A -85,B 0,C 180,E1 -7512.571,E2 -7512.571} C_VEL
LIN {X 0,Y 467.566,Z 511.238,A -85,B 0,C 180,E1 -7516.176,E2 -7516.176} C_VEL
LIN {X 0,Y 467.581,Z 511.24,A -85,B 0,C 180,E1 -7518.721,E2 -7518.721} C_VEL
LIN {X 0,Y 467.57,Z 511.241,A -85,B 0,C 180,E1 -7521.406,E2 -7521.406} C_VEL
LIN {X 0,Y 467.555,Z 511.24,A -85,B 0,C 180,E1 -7524.26,E2 -7524.26} C_VEL
